         DBX222_6 : Bool;
         DBX222_7 : Bool;
         DBX223_0 : Bool;
         DBX223_1 : Bool;
         DBX223_2 : Bool;
         DBX223_3 : Bool;
         DBX223_4 : Bool;
         DBX223_5 : Bool;
         DBX223_6 : Bool;
         DBX223_7 : Bool;
         DBX224_0 : Bool;
         DBX224_1 : Bool;
         DBX224_2 : Bool;
         DBX224_3 : Bool;
         DBX224_4 : Bool;
         DBX224_5 : Bool;
         DBX224_6 : Bool;
         DBX224_7 : Bool;
         DBX225_0 : Bool;
         DBX225_1 : Bool;
         DBX225_2 : Bool;
         DBX225_3 : Bool;
         DBX225_4 : Bool;
         DBX225_5 : Bool;
         DBX225_6 : Bool;
         DBX225_7 : Bool;
         DBX226_0 : Bool;   // 9;CHAIN T7B;Stop Permisie Cuplare Lant T7-B Actionat;DI;A1;26;M;K
         DBX226_1 : Bool;   // 9;CHAIN T7B;TimeOut Cuplare/Decuplare Alim.Inv. Lant T7-B;DI;A1;26;M;O;K
         DBX226_2 : Bool;   // 9;CHAIN T7B;Lipsa Tensiune de Comanda Lant T7-B;DI;A1;26;M;K
         DBX226_3 : Bool;   // 9;CHAIN T7B;Sectionator Alim.Inv. Mot. Lant T7-B Decuplat;DI;A2;26;M;K
         DBX226_4 : Bool;   // 9;CHAIN T7B;Inverter Mot. Lant T7-B Avarie;DI;A2;26;M;O;K
         DBX226_5 : Bool;
         DBX226_6 : Bool;
         DBX226_7 : Bool;
         DBX227_0 : Bool;
         DBX227_1 : Bool;   // 9;CHAIN T7B;TimeOut Deplasare Lant T7-B in pozitia Pas;DI;A1;26;M;O;K
         DBX227_2 : Bool;   // 9;CHAIN T7B;Problema Contactor sau Prot. Termica Frana Lant T7-B;DI;A1;26;M;K
         DBX227_3 : Bool;   // 9;CHAIN T7B;TimeOut Deplasare Lant T7-B;DI;A1;26;M;O;K
         DBX227_4 : Bool;   // 9;CHAIN T7B;Disj. Termic Alim. Vent.Mot. Lant T7-B Declansat;DI;A1;26;M
         DBX227_5 : Bool;
         DBX227_6 : Bool;
         DBX227_7 : Bool;
         DBX228_0 : Bool;
         DBX228_1 : Bool;
         DBX228_2 : Bool;
         DBX228_3 : Bool;
         DBX228_4 : Bool;
         DBX228_5 : Bool;
         DBX228_6 : Bool;
         DBX228_7 : Bool;
         DBX229_0 : Bool;
         DBX229_1 : Bool;
         DBX229_2 : Bool;
         DBX229_3 : Bool;
         DBX229_4 : Bool;
         DBX229_5 : Bool;
         DBX229_6 : Bool;
         DBX229_7 : Bool;
         DBX230_0 : Bool;   // 9;FLIPPER2 T7B;Lipsa Tensiune Alimentare Aruncator 2 T7-B;DI;A1;26;M;K
         DBX230_1 : Bool;   // 9;FLIPPER2 T7B;TimeOut Deplasare Aruncator 2 T7-B in pozitia Sus;DI;A1;26;M;O
         DBX230_2 : Bool;   // 9;FLIPPER2 T7B;TimeOut Deplasare Aruncator 2 T7-B in pozitia Jos;DI;A1;26;M;O
         DBX230_3 : Bool;
         DBX230_4 : Bool;
         DBX230_5 : Bool;
         DBX230_6 : Bool;
         DBX230_7 : Bool;
         DBX231_0 : Bool;
         DBX231_1 : Bool;
         DBX231_2 : Bool;
         DBX231_3 : Bool;
         DBX231_4 : Bool;
         DBX231_5 : Bool;
         DBX231_6 : Bool;
         DBX231_7 : Bool;
         DBX232_0 : Bool;
         DBX232_1 : Bool;
         DBX232_2 : Bool;
         DBX232_3 : Bool;
         DBX232_4 : Bool;
         DBX232_5 : Bool;
         DBX232_6 : Bool;
         DBX232_7 : Bool;
         DBX233_0 : Bool;
         DBX233_1 : Bool;
         DBX233_2 : Bool;
         DBX233_3 : Bool;
         DBX233_4 : Bool;
         DBX233_5 : Bool;
         DBX233_6 : Bool;
         DBX233_7 : Bool;
         DBX234_0 : Bool;   // 9;COLLECTOR T7B;Disjunctor Termic Motor Colector T7-B;DI;A1;26;M
         DBX234_1 : Bool;   // 9;COLLECTOR T7B;TimeOut Deplasare Colector T7-B;DI;A1;26;M;O
         DBX234_2 : Bool;   // 9;COLLECTOR T7B;Disjunctor Termic Alim. Motor Colector T7-B;DI;A1;26;M
         DBX234_3 : Bool;   // 9;COLLECTOR T7B;Colector T7-B LB PLIN OFF;SQ;W3;26;O
         DBX234_4 : Bool;
         DBX234_5 : Bool;
         DBX234_6 : Bool;
         DBX234_7 : Bool;
         DBX235_0 : Bool;
         DBX235_1 : Bool;
         DBX235_2 : Bool;
         DBX235_3 : Bool;
         DBX235_4 : Bool;
         DBX235_5 : Bool;
         DBX235_6 : Bool;
         DBX235_7 : Bool;
         DBX236_0 : Bool;
         DBX236_1 : Bool;
         DBX236_2 : Bool;
         DBX236_3 : Bool;
         DBX236_4 : Bool;
         DBX236_5 : Bool;
         DBX236_6 : Bool;
         DBX236_7 : Bool;
         DBX237_0 : Bool;
         DBX237_1 : Bool;
         DBX237_2 : Bool;
         DBX237_3 : Bool;
         DBX237_4 : Bool;
         DBX237_5 : Bool;
         DBX237_6 : Bool;
         DBX237_7 : Bool;
         DBX238_0 : Bool;
         DBX238_1 : Bool;
         DBX238_2 : Bool;
         DBX238_3 : Bool;
         DBX238_4 : Bool;
         DBX238_5 : Bool;
         DBX238_6 : Bool;
         DBX238_7 : Bool;
         DBX239_0 : Bool;
         DBX239_1 : Bool;
         DBX239_2 : Bool;
         DBX239_3 : Bool;
         DBX239_4 : Bool;
         DBX239_5 : Bool;
         DBX239_6 : Bool;
         DBX239_7 : Bool;
         DBX240_0 : Bool;
         DBX240_1 : Bool;
         DBX240_2 : Bool;
         DBX240_3 : Bool;
         DBX240_4 : Bool;
         DBX240_5 : Bool;
         DBX240_6 : Bool;
         DBX240_7 : Bool;
         DBX241_0 : Bool;
         DBX241_1 : Bool;
         DBX241_2 : Bool;
         DBX241_3 : Bool;
         DBX241_4 : Bool;
         DBX241_5 : Bool;
         DBX241_6 : Bool;
         DBX241_7 : Bool;
         DBX242_0 : Bool;   // 9;ROLLS T7-C;Suma Disj. Termice Mot. C.Role T7-C Declansat;DI;A1;25;M;K
         DBX242_1 : Bool;   // 9;ROLLS T7-C;Sectionator Alim.Inv. Mot. C.Role T7-C Decuplat;DI;A2;25;M
         DBX242_2 : Bool;   // 9;ROLLS T7-C;Lipsa Tensiune de Comanda C.Role T7-C;DI;A1;25;M
         DBX242_3 : Bool;   // 9;ROLLS T7-C;TimeOut Rotire Role C.Role T7-C;DI;A1;25;M;O
         DBX242_4 : Bool;   // 9;ROLLS T7-C;Role T7-C TimeOut Teava ON;SQ;A1;25;O
         DBX242_5 : Bool;   // 9;ROLLS T7-C;Role T7-C TimeOut Teava SLOW;SQ;A1;25;O
         DBX242_6 : Bool;   // 9;ROLLS T7-C;Role T7-C TimeOut Pozitionare Teava;SQ;A1;25;O
         DBX242_7 : Bool;   // 9;ROLLS T7-C;Role T7-C TimeOut Teava OFF;SQ;A1;25;O
         DBX243_0 : Bool;
         DBX243_1 : Bool;
         DBX243_2 : Bool;
         DBX243_3 : Bool;
         DBX243_4 : Bool;   // 9;ROLLS T7-C;Disj. Termic Alim.Vent.Mot. C.Role T7-C - Declansat;DI;A1;25;M
         DBX243_5 : Bool;
         DBX243_6 : Bool;   // 9;ROLLS T7-C;Inverter Mot. C.Role T7-C - Avarie;DI;A1;25;M;O
         DBX243_7 : Bool;
         DBX244_0 : Bool;
         DBX244_1 : Bool;
         DBX244_2 : Bool;   // 9;ROLLS T7-C;Suma Disj. Th. Vent.Mot. C.Role T7-C - Declansat;DI;A1;25;M
         DBX244_3 : Bool;   // 9;ROLLS T7-C;TimeOut Cuplare/Decuplare Vent.Mot. C.Role T7-C;DI;A1;25;M;O
         DBX244_4 : Bool;   // 9;ROLLS T7-C;TimeOut Cuplare/Decuplare Alim.Inv. C.Role T7-C;DI;A1;25;M;O
         DBX244_5 : Bool;
         DBX244_6 : Bool;
         DBX244_7 : Bool;
         DBX245_0 : Bool;
         DBX245_1 : Bool;
         DBX245_2 : Bool;
         DBX245_3 : Bool;
         DBX245_4 : Bool;
         DBX245_5 : Bool;
         DBX245_6 : Bool;
         DBX245_7 : Bool;
         DBX246_0 : Bool;   // 9;FLIPPER T7-C;Lipsa Tensiune Alimentare Aruncator T7-C;DI;A1;25;M
         DBX246_1 : Bool;   // 9;FLIPPER T7-C;TimeOut Deplasare Aruncator T7-C in pozitia Sus;DI;A1;25;M;O
         DBX246_2 : Bool;   // 9;FLIPPER T7-C;TimeOut Deplasare Aruncator T7-C in pozitia Jos;DI;A1;25;M;O
         DBX246_3 : Bool;
         DBX246_4 : Bool;
         DBX246_5 : Bool;
         DBX246_6 : Bool;
         DBX246_7 : Bool;
         DBX247_0 : Bool;
         DBX247_1 : Bool;
         DBX247_2 : Bool;
         DBX247_3 : Bool;
         DBX247_4 : Bool;
         DBX247_5 : Bool;
         DBX247_6 : Bool;
         DBX247_7 : Bool;
         DBX248_0 : Bool;
         DBX248_1 : Bool;
         DBX248_2 : Bool;
         DBX248_3 : Bool;
         DBX248_4 : Bool;
         DBX248_5 : Bool;
         DBX248_6 : Bool;
         DBX248_7 : Bool;
         DBX249_0 : Bool;
         DBX249_1 : Bool;
         DBX249_2 : Bool;
         DBX249_3 : Bool;
         DBX249_4 : Bool;
         DBX249_5 : Bool;
         DBX249_6 : Bool;
         DBX249_7 : Bool;
         DBX250_0 : Bool;   // 9;COLLECTOR T7C;Disjunctor Termic Motor Colector T7-C;DI;A1;25;M
         DBX250_1 : Bool;   // 9;COLLECTOR T7C;TimeOut Deplasare Colector T7-C;DI;A1;25;M;O
         DBX250_2 : Bool;   // 9;COLLECTOR T7C;Disjunctor Termic Alim. Motor Colector T7-C;DI;A1;25;M
         DBX250_3 : Bool;   // 9;COLLECTOR T7C;Colector T7-C TimeOut Colector Plin;SQ;A1;25;O
         DBX250_4 : Bool;
         DBX250_5 : Bool;
         DBX250_6 : Bool;
         DBX250_7 : Bool;
         DBX251_0 : Bool;
         DBX251_1 : Bool;
         DBX251_2 : Bool;
         DBX251_3 : Bool;
         DBX251_4 : Bool;
         DBX251_5 : Bool;
         DBX251_6 : Bool;
         DBX251_7 : Bool;
         DBX252_0 : Bool;
         DBX252_1 : Bool;
         DBX252_2 : Bool;
         DBX252_3 : Bool;
         DBX252_4 : Bool;
         DBX252_5 : Bool;
         DBX252_6 : Bool;
         DBX252_7 : Bool;
         DBX253_0 : Bool;
         DBX253_1 : Bool;
         DBX253_2 : Bool;
         DBX253_3 : Bool;
         DBX253_4 : Bool;
         DBX253_5 : Bool;
         DBX253_6 : Bool;
         DBX253_7 : Bool;
         DBX254_0 : Bool;   // 9;TAMPON T7-C;Lipsa Tensiune Alimentare Tampon T7-C;DI;A1;25;M
         DBX254_1 : Bool;   // 9;TAMPON T7-C;TimeOut Deplasare Tampon T7-C in pozitia Sus;DI;A1;25;M;O
         DBX254_2 : Bool;   // 9;TAMPON T7-C;TimeOut Deplasare Tampon T7-C in pozitia Jos;DI;A1;25;M;O
         DBX254_3 : Bool;
         DBX254_4 : Bool;
         DBX254_5 : Bool;
         DBX254_6 : Bool;
         DBX254_7 : Bool;
         DBX255_0 : Bool;
         DBX255_1 : Bool;
         DBX255_2 : Bool;
         DBX255_3 : Bool;
         DBX255_4 : Bool;
         DBX255_5 : Bool;
         DBX255_6 : Bool;
         DBX255_7 : Bool;
         DBX256_0 : Bool;
         DBX256_1 : Bool;
         DBX256_2 : Bool;
         DBX256_3 : Bool;
         DBX256_4 : Bool;
         DBX256_5 : Bool;
         DBX256_6 : Bool;
         DBX256_7 : Bool;
         DBX257_0 : Bool;
         DBX257_1 : Bool;
         DBX257_2 : Bool;
         DBX257_3 : Bool;
         DBX257_4 : Bool;
         DBX257_5 : Bool;
         DBX257_6 : Bool;
         DBX257_7 : Bool;
         DBX258_0 : Bool;
         DBX258_1 : Bool;
         DBX258_2 : Bool;
         DBX258_3 : Bool;
         DBX258_4 : Bool;
         DBX258_5 : Bool;
         DBX258_6 : Bool;
         DBX258_7 : Bool;
         DBX259_0 : Bool;
         DBX259_1 : Bool;
         DBX259_2 : Bool;
         DBX259_3 : Bool;
         DBX259_4 : Bool;
         DBX259_5 : Bool;
         DBX259_6 : Bool;
         DBX259_7 : Bool;
         DBX260_0 : Bool;   // 9;DEBITARE;Disjunctor Termic Alim. Convertizor Lama;DI;A1;25;M
         DBX260_1 : Bool;   // 9;DEBITARE;TimeOut Cuplare/Decup. Cont. Convertizor Lama;DI;A1;25;M;O
         DBX260_2 : Bool;   // 9;DEBITARE;Disjunctor Termic Alim. Pompa Statie Hidraulica;DI;A2;25;M
         DBX260_3 : Bool;   // 9;DEBITARE;TimeOut Cuplare/Decup. Pompa Statie Hidraulica;DI;A1;25;M;O
         DBX260_4 : Bool;   // 9;DEBITARE;Disjunctor Termic Alim. Rezistenta Incalzire Ulei;DI;A1;25;M
         DBX260_5 : Bool;   // 9;DEBITARE;TimeOut Cuplare/Decup. Rezistenta Incalzire Ulei;DI;A1;25;M;O
         DBX260_6 : Bool;   // 9;DEBITARE;Disjunctor Termic Alim. Motor Vent. Statie Hidr.;DI;A1;25;M
         DBX260_7 : Bool;   // 9;DEBITARE;TimeOut Cuplare/Decup. Motor Vent. Statie Hidr.;DI;A1;25;M;O
         DBX261_0 : Bool;   // 9;DEBITARE;Disjunctor Termic Alim. Motor Pompa Racire Lama;DI;A1;25;M
         DBX261_1 : Bool;   // 9;DEBITARE;TimeOut Cuplare/Decup. Motor Pompa Racire Lama;DI;A1;25;M;O
         DBX261_2 : Bool;   // 9;DEBITARE;TimeOut Depl. Rola Singulara T7C in Pozitia 'Sus';DI;A1;25;M;O
         DBX261_3 : Bool;   // 9;DEBITARE;TimeOut Depl. Rola Singulara T7C in Pozitia 'Jos';DI;A1;25;M;O
         DBX261_4 : Bool;   // 9;DEBITARE;TimeOut Depl. Role T7C in Pozitia 'Sus';DI;A1;25;M;O
         DBX261_5 : Bool;   // 9;DEBITARE;TimeOut Depl. Role T7C in Pozitia 'Jos';DI;A1;25;M;O
         DBX261_6 : Bool;   // 9;DEBITARE;TimeOut Depl. Opritor Mobil in Pozitia 'Sus';DI;A1;25;M;O
         DBX261_7 : Bool;   // 9;DEBITARE;TimeOut Depl. Opritor Mobil in Pozitia 'Jos';DI;A1;25;M;O
         DBX262_0 : Bool;   // 9;DEBITARE;TimeOut Depl. Lama Circulara in Pozitia 'Sus';DI;A1;25;M;O
         DBX262_1 : Bool;   // 9;DEBITARE;TimeOut Depl. Lama Circulara in Pozitia 'Jos';DI;A1;25;M;O
         DBX262_2 : Bool;   // 9;DEBITARE;TimeOut Depl. Menghina in Pozitia 'Deschis';DI;A1;25;M;O
         DBX262_3 : Bool;   // 9;DEBITARE;Avertizare Coliziune Teava cu Rola Singulara T7C;DI;A1;25;O
         DBX262_4 : Bool;   // 9;DEBITARE;Avertizare Coliziune Teava cu Calea cu Role T7C;DI;A1;25;O
         DBX262_5 : Bool;   // 9;DEBITARE;Avertizare Coliziune Teava Opritor Mobil Masa T7C;DI;A1;25;O
         DBX262_6 : Bool;   // 9;DEBITARE;Avertizare Coliziune Teava cu Lama Circulara T7C;DI;A1;25;O
         DBX262_7 : Bool;   // 9;DEBITARE;Stare Convertizor - Avarie;DI;A1;25;M;O
         DBX263_0 : Bool;   // 9;DEBITARE;Disjuntor Termic Motor Lama Circulara - Declansat;DI;A1;25;M
         DBX263_1 : Bool;   // 9;DEBITARE;Nivel Apa Bazin Racire - Minim;DI;A1;25;M;O
         DBX263_2 : Bool;   // 9;DEBITARE;Temperatura Ulei Hidraulic - Minim;DI;W2;25;M;O
         DBX263_3 : Bool;   // 9;DEBITARE;Temperatura Ulei Hidraulic - Ridicat;DI;W2;25;M;O
         DBX263_4 : Bool;   // 9;DEBITARE;Temperatura Ulei Hidraulic - Maxim;DI;A1;25;M;O
         DBX263_5 : Bool;   // 9;DEBITARE;Nivel Ulei Hidraulic - Minim;DI;A1;25;M;O
         DBX263_6 : Bool;   // 9;DEBITARE;Releu Avarie (ciuperca) - Declansat;EM;A1;25;M;O;K
         DBX263_7 : Bool;
         DBX264_0 : Bool;   // 4;FIERASTRAU KASTO;Fierastrau Kasto Emergenta Apasata;EM;A1;11;M;O;K
         DBX264_1 : Bool;   // 4;FIERASTRAU KASTO;Avarie/Avertizare Fierastrau Kasto;DI;A1;11;M;O
         DBX264_2 : Bool;   // 4;FIERASTRAU KASTO;Pupitru Cabina Emergenta Apasata;EM;A1;11;M;O;K
         DBX264_3 : Bool;   // 4;TAMPON MASURARE PROBA;Disjunctor motor regl. proba decupl.;DI;A1;11;M
         DBX264_4 : Bool;   // 4;TAMPON MASURARE PROBA;Lipsa fbk cont linie mot. misc. inainte;DI;A1;11;M
         DBX264_5 : Bool;   // 4;TAMPON MASURARE PROBA;Lipsa fbk cont linie mot. misc. inapoi;DI;A1;11;M
         DBX264_6 : Bool;   // 4;ROLE KASTO;Disjunctor protectie ventilator motor 1 cuplat;DI;W2;11;M
         DBX264_7 : Bool;   // 4;ROLE KASTO;Confirmare cuplare contactor ventilator1 cuplat;DI;W2;11;M
         DBX265_0 : Bool;   // 4;ROLE KASTO;Disjunctor protectie ventilator motor 2 cuplat;DI;W2;11;M
         DBX265_1 : Bool;   // 4;ROLE KASTO;Confirmare cuplare contactor ventilator2 cuplat;DI;W2;11;M
         DBX265_2 : Bool;   // 4;ROLE KASTO;Disjunctor protectie ventilator motor 3 cuplat;DI;W2;11;M
         DBX265_3 : Bool;   // 4;ROLE KASTO;Confirmare cuplare contactor ventilator3 cuplat;DI;W2;11;M
         DBX265_4 : Bool;   // 4;ROLE KASTO;Disjunctor protectie ventilator motor 4 cuplat;DI;W2;11;M
         DBX265_5 : Bool;   // 4;ROLE KASTO;Confirmare cuplare contactor ventilator4 cuplat;DI;W2;11;M
         DBX265_6 : Bool;   // 4;ROLE KASTO;Disjunctor protectie ventilator motor 5 cuplat;DI;W2;11;M
         DBX265_7 : Bool;   // 4;ROLE KASTO;Confirmare cuplare contactor ventilator5 cuplat;DI;W2;11;M
         DBX266_0 : Bool;   // 4;ROLE KASTO;Disjunctor protectie ventilator motor 6 cuplat;DI;W2;11;M
         DBX266_1 : Bool;   // 4;ROLE KASTO;Confirmare cuplare contactor ventilator6 cuplat;DI;W2;11;M
         DBX266_2 : Bool;   // 4;ROLE KASTO;Disjunctor protectie ventilator motor 7 cuplat;DI;W2;11;M
         DBX266_3 : Bool;   // 4;ROLE KASTO;Confirmare cuplare contactor ventilator7 cuplat;DI;W2;11;M
         DBX266_4 : Bool;   // 4;ROLE KASTO;Disjunctor protectie ventilator motor 8 cuplat;DI;W2;11;M
         DBX266_5 : Bool;   // 4;ROLE KASTO;Confirmare cuplare contactor ventilator8 cuplat;DI;W2;11;M
         DBX266_6 : Bool;   // 4;ROLE KASTO;Disjunctor protectie ventilator motor 9 cuplat;DI;W2;11;M
         DBX266_7 : Bool;   // 4;ROLE KASTO;Confirmare cuplare contactor ventilator9 cuplat;DI;W2;11;M
         DBX267_0 : Bool;   // 4;ROLE KASTO;Disjunctor protectie ventilator motor 10 cuplat;DI;W2;11;M
         DBX267_1 : Bool;   // 4;ROLE KASTO;Confirmare cuplare contactor ventilat.10 cuplat;DI;W2;11;M
         DBX267_2 : Bool;   // 4;ROLE KASTO;Disjunctor protectie ventilator motor 11 cuplat;DI;W2;11;M
         DBX267_3 : Bool;   // 4;ROLE KASTO;Confirmare cuplare contactor ventilat.11 cuplat;DI;W2;11;M
         DBX267_4 : Bool;   // 4;ROLE KASTO;Disjunctor protectie ventilator motor 12 cuplat;DI;W2;11;M
         DBX267_5 : Bool;   // 4;ROLE KASTO;Confirmare cuplare contactor ventilat.12 cuplat;DI;W2;11;M
         DBX267_6 : Bool;   // 4;ROLE KASTO;Disjunctor protectie ventilator motor 13 cuplat;DI;W2;11;M
         DBX267_7 : Bool;   // 4;ROLE KASTO;Confirmare cuplare contactor ventilat.13 cuplat;DI;W2;11;M
         DBX268_0 : Bool;   // 4;ROLE KASTO;Disjunctor protectie ventilator motor 14 cuplat;DI;W2;11;M
         DBX268_1 : Bool;   // 4;ROLE KASTO;Confirmare cuplare contactor ventilat.14 cuplat;DI;W2;11;M
         DBX268_2 : Bool;   // 4;ROLE KASTO;Disjunctor protectie ventilator motor 15 cuplat;DI;W2;11;M
         DBX268_3 : Bool;   // 4;ROLE KASTO;Confirmare cuplare contactor ventilat.15 cuplat;DI;W2;11;M
         DBX268_4 : Bool;   // 4;ROLE KASTO;Fuzibil protectie convertizor;DI;A1;11;M
         DBX268_5 : Bool;   // 4;ROLE KASTO;Disjunctor monitorizare fuzibil convertizor;DI;A1;11;M
         DBX268_6 : Bool;   // 4;ROLE KASTO;Contactor alimentare convertizor;DI;A1;11;M
         DBX268_7 : Bool;   // 4;ROLE KASTO;Disjunctor protectie motoare;DI;A1;11;M
         DBX269_0 : Bool;   // 4;ROLE KASTO;Rola Mobila nu este ridicata;DI;A1;11;M
         DBX269_1 : Bool;
         DBX269_2 : Bool;
         DBX269_3 : Bool;
         DBX269_4 : Bool;
         DBX269_5 : Bool;
         DBX269_6 : Bool;
         DBX269_7 : Bool;
         DBX270_0 : Bool;   // 9;MARCARE;Disjunctor decuplat;DI;A2;24;M;K
         DBX270_1 : Bool;   // 9;MARCARE;Contactor ridicare decuplat;DI;A2;24;M;K
         DBX270_2 : Bool;   // 9;MARCARE;Contactor coborare decuplat;DI;A2;24;M;K
         DBX270_3 : Bool;   // 9;MARCARE;OCV camera fault;DI;A1;24;O
         DBX270_4 : Bool;   // 9;MARCARE;OCV alarma scor;DI;A1;24;O
         DBX270_5 : Bool;
         DBX270_6 : Bool;
         DBX270_7 : Bool;
         DBX271_0 : Bool;   // 4;FIERASTRAU KASTO;Citire atribute - Level 2 avarie generala;TK;W2;11;O
         DBX271_1 : Bool;   // 4;FIERASTRAU KASTO;Citire atribute - Destinatie plina;TK;W2;11;O
         DBX271_2 : Bool;   // 4;FIERASTRAU KASTO;Citire atribute - Sursa goala;TK;W2;11;O
         DBX271_3 : Bool;   // 4;FIERASTRAU KASTO;Incarca zona - Level 2 avarie generala;TK;W2;11;O
         DBX271_4 : Bool;   // 4;FIERASTRAU KASTO;Incarca zona - idTrackingItem invalid;TK;W2;11;O
         DBX271_5 : Bool;   // 4;FIERASTRAU KASTO;Incarca zona-Itemul nu e in prima pozitie;TK;W2;11;O
         DBX271_6 : Bool;   // 4;FIERASTRAU KASTO;Incarca zona - Destinatie plina;TK;W2;11;O
         DBX271_7 : Bool;   // 4;FIERASTRAU KASTO;Incarca zona - Sursa goala;TK;W2;11;O
         DBX272_0 : Bool;   // 4;FIERASTRAU KASTO;Verifica zona T4-2-Level2 avarie generala;TK;W2;11;O
         DBX272_1 : Bool;   // 4;FIERASTRAU KASTO;Descarca zona Kasto-Level2 avarie general;TK;W2;11;O
         DBX272_2 : Bool;   // 4;FIERASTRAU KASTO;Descarca zona Kasto - Destinatie plina;TK;W2;11;O
         DBX272_3 : Bool;   // 4;FIERASTRAU KASTO;Descarca zona Kasto - Sursa goala;TK;W2;11;O
         DBX272_4 : Bool;   // 4;FIERASTRAU KASTO;Verifica zona Kasto-Level2 avarie general;TK;W2;11;O
         DBX272_5 : Bool;   // 4;FIERASTRAU KASTO;Pat racire - Zona Kasto pachete diferite;TK;W2;11;O
         DBX272_6 : Bool;
         DBX272_7 : Bool;
         DBX273_0 : Bool;
         DBX273_1 : Bool;
         DBX273_2 : Bool;
         DBX273_3 : Bool;
         DBX273_4 : Bool;
         DBX273_5 : Bool;
         DBX273_6 : Bool;
         DBX273_7 : Bool;
         DBX274_0 : Bool;
         DBX274_1 : Bool;
         DBX274_2 : Bool;
         DBX274_3 : Bool;
         DBX274_4 : Bool;
         DBX274_5 : Bool;
         DBX274_6 : Bool;
         DBX274_7 : Bool;
         DBX275_0 : Bool;
         DBX275_1 : Bool;
         DBX275_2 : Bool;
         DBX275_3 : Bool;
         DBX275_4 : Bool;
         DBX275_5 : Bool;
         DBX275_6 : Bool;
         DBX275_7 : Bool;
         DBX276_0 : Bool;
         DBX276_1 : Bool;
         DBX276_2 : Bool;
         DBX276_3 : Bool;
         DBX276_4 : Bool;
         DBX276_5 : Bool;
         DBX276_6 : Bool;
         DBX276_7 : Bool;
         DBX277_0 : Bool;
         DBX277_1 : Bool;
         DBX277_2 : Bool;
         DBX277_3 : Bool;
         DBX277_4 : Bool;
         DBX277_5 : Bool;
         DBX277_6 : Bool;
         DBX277_7 : Bool;
         DBX278_0 : Bool;
         DBX278_1 : Bool;
         DBX278_2 : Bool;
         DBX278_3 : Bool;
         DBX278_4 : Bool;
         DBX278_5 : Bool;
         DBX278_6 : Bool;
         DBX278_7 : Bool;
         DBX279_0 : Bool;
         DBX279_1 : Bool;
         DBX279_2 : Bool;
         DBX279_3 : Bool;
         DBX279_4 : Bool;
         DBX279_5 : Bool;
         DBX279_6 : Bool;
         DBX279_7 : Bool;
         DBX280_0 : Bool;   // 1;Create Tracking;Time Out LEV2;TK;W2;1;O
         DBX280_1 : Bool;   // 1;New item load;Time Out LEV2;TK;W2;1;O
         DBX280_2 : Bool;   // 1;Item Count;Time Out LEV2;TK;W2;1;O
         DBX280_3 : Bool;   // 2;Check Product;Time Out LEV2;TK;W2;1;O
         DBX280_4 : Bool;   // 4;Check Product;Time Out LEV2;TK;W2;8;O
         DBX280_5 : Bool;   // 5;Create Tracking;Time Out LEV2;TK;W2;16;O
         DBX280_6 : Bool;   // 5;M5 Temper Entrance Check Product;Time Out LEV2;TK;W2;15;O
         DBX280_7 : Bool;   // 5;M5 Temper Entrance New Item Load;Time Out LEV2;TK;W2;15;O
         DBX281_0 : Bool;   // 5;M5 Temper Entrance Item Count;Time Out LEV2;TK;W2;15;O
         DBX281_1 : Bool;   // 6;M6 Temper Furnace Check Product;Time Out LEV2;TK;W2;15;O
         DBX281_2 : Bool;   // 8;M8 Straightening Check Product;Time Out LEV2;TK;W2;22;O
         DBX281_3 : Bool;   // 8;M8 Straightening New Item Load;Time Out LEV2;TK;W2;22;O
         DBX281_4 : Bool;   // 8;M8 Straightening New Item Count;Time Out LEV2;TK;W2;22;O
         DBX281_5 : Bool;   // 9;M9 Stamping Check Product;Time Out LEV2;TK;W2;23;O
         DBX281_6 : Bool;   // 9;M9 Stamping New Item Load;Time Out LEV2;TK;W2;23;O
         DBX281_7 : Bool;   // 9;M9 Stamping Item Count;Time Out LEV2;TK;W2;23;O
         DBX282_0 : Bool;   // 10;M10 Exit Check Product;Time Out LEV2;TK;W2;26;O
         DBX282_1 : Bool;   // 10;M10 Exit New Item Load;Time Out LEV2;TK;W2;26;O
         DBX282_2 : Bool;   // 10;M10 Exit New Item Count;Time Out LEV2;TK;W2;26;O
         DBX282_3 : Bool;   // 1;Z1 Entrance Quench Load;Time Out LEV2;TK;W2;1;O
         DBX282_4 : Bool;   // 3;Z3 Quenching Head Unload;Time Out LEV2;TK;W2;8;O
         DBX282_5 : Bool;   // 3;Z4 Exit Quench Unload;Time Out LEV2;TK;W2;10;O
         DBX282_6 : Bool;   // 4;Z5 Cool. Bench T4 load;Time Out LEV2;TK;W2;10;O
         DBX282_7 : Bool;   // 4;Z5 Cool. Bench T4 Exit Check;Time Out LEV2;TK;W2;10;O
         DBX283_0 : Bool;   // 4;Z5 Cool. Bench T4 Unload;Time Out LEV2;TK;W2;10;O
         DBX283_1 : Bool;   // 4;Z6 Exit T4 Get Pipe Attributes;Time Out LEV2;TK;W2;10;O
         DBX283_2 : Bool;   // 4;Z6 Exit T4 Unload;Time Out LEV2;TK;W2;14;O
         DBX283_3 : Bool;   // 4;Z8 Cool. Bench T5 Exit Load;Time Out LEV2;TK;W2;14;O
         DBX283_4 : Bool;   // 4;Z8 Cool. Bench T5 Exit Check;Time Out LEV2;TK;W2;14;O
         DBX283_5 : Bool;   // 4;Z8 Cool. Bench T5 Unload;Time Out LEV2;TK;W2;14;O
         DBX283_6 : Bool;   // 4;Z9 Exit T5 Get Pipe Attributes;Time Out LEV2;TK;W2;14;O
         DBX283_7 : Bool;   // 1;Z1 Entrance Quench Exit Check;Time Out LEV2;TK;W2;1;O
         DBX284_0 : Bool;   // 4;Z9 Exit T5 Unload;Time Out LEV2;TK;W2;15;O
         DBX284_1 : Bool;   // 4;Z10 Cool. Bench T6 Exit Load;Time Out LEV2;TK;W2;15;O
         DBX284_2 : Bool;   // 4;Z10 Cool. Bench T6 Exit Check;Time Out LEV2;TK;W2;15;O
         DBX284_3 : Bool;   // 4;Z10 Cool. Bench T6 Unload;Time Out LEV2;TK;W2;15;O
         DBX284_4 : Bool;   // 5;Z11 Entrance Temper Zone Load;Time Out LEV2;TK;W2;16;O
         DBX284_5 : Bool;   // 5;Z11 Entrance Temper Get Pipe Attributes;Time Out LEV2;TK;W2;15;O
         DBX284_6 : Bool;   // 7;Z13 Exit Temper Unload;Time Out LEV2;TK;W2;21;O
         DBX284_7 : Bool;   // 8;Z14 T7 Unload;Time Out LEV2;TK;W2;21;O
         DBX285_0 : Bool;   // 8;Z15 Straightening Unload;Time Out LEV2;TK;W2;22;O
         DBX285_1 : Bool;   // 8;Z16 T7A Loading Unload;Time Out LEV2;TK;W2;23;O
         DBX285_2 : Bool;   // 8;Z17 Cool.Bench T7A Exit Load;Time Out LEV2;TK;W2;23;O
         DBX285_3 : Bool;   // 8;Z17 Cool.Bench T7A Exit Check;Time Out LEV2;TK;W2;23;O
         DBX285_4 : Bool;   // 8;Z17 Cool.Bench T7A Unload;Time Out LEV2;TK;W2;23;O
         DBX285_5 : Bool;   // 9;Z18 Exit T7A Exit Check;Time Out LEV2;TK;W2;23;O
         DBX285_6 : Bool;   // 9;Z18 Exit T7A Unload;Time Out LEV2;TK;W2;26;O
         DBX285_7 : Bool;   // 9;Z18 Exit T7A Get Pipe Attributes;Time Out LEV2;TK;W2;23;O
         DBX286_0 : Bool;   // 9;Z19 Temper Sample Cut Load;Time Out LEV2;TK;W2;25;O
         DBX286_1 : Bool;   // 9;Z19 Temper Sample Cut Unload;Time Out LEV2;TK;W2;25;O
         DBX286_2 : Bool;   // 9;Z20 Cool.Bench T7B Exit Load;Time Out LEV2;TK;W2;26;O
         DBX286_3 : Bool;   // 9;Z20 Cool.Bench T7B Exit Check;Time Out LEV2;TK;W2;26;O
         DBX286_4 : Bool;   // 9;Z20 Cool.Bench T7B Unload;Time Out LEV2;TK;W2;26;O
         DBX286_5 : Bool;   // 9;Z21 Exit T7B Check;Time Out LEV2;TK;W2;26;O
         DBX286_6 : Bool;   // 9;Z21 Exit T7B Unload;Time Out LEV2;TK;W2;26;O
         DBX286_7 : Bool;   // 9;Send Data Stamping Machine;Time Out LEV2;TK;W2;23;O
         DBX287_0 : Bool;   // 8;Z14 T7 Exit Check;Time Out LEV2;TK;W2;21;O
         DBX287_1 : Bool;   // 3;Z3 Quenching Head Exit Check;Time Out LEV2;TK;W2;8;O
         DBX287_2 : Bool;   // 5;Z11 Temper Entrance Exit Check;Time Out LEV2;TK;W2;16;O
         DBX287_3 : Bool;   // 4;Z7 Quench Sample Unload;Time Out LEV2;TK;W2;12;O
         DBX287_4 : Bool;   // 4;Z23 Load T5 Zone Unload;Time Out LEV2;TK;W2;14;O
         DBX287_5 : Bool;   // 4;Z6 Exit T4 Load;Time Out LEV2;TK;W2;14;O
         DBX287_6 : Bool;   // 9;Z24 Load T7-B Zone Unload;Time Out LEV2;TK;W2;26;O
         DBX287_7 : Bool;   // 9;Z18 Exit T7-A Load;Time Out LEV2;TK;W2;23;O
         DBX288_0 : Bool;   // 9;Z24 Load T7-B Get Pipe Attributes;Time Out LEV2;TK;W2;26;O
         DBX288_1 : Bool;   // 4;Z6 Exit T4 Exit Check;Time Out LEV2;TK;W2;10;O
         DBX288_2 : Bool;   // 4;Z23 Load T5 Exit Check;Time Out LEV2;TK;W2;14;O
         DBX288_3 : Bool;   // 4;Z9 Exit T5 Exit Check;Time Out LEV2;TK;W2;14;O
         DBX288_4 : Bool;   // 9;Z24 Load T7B Exit Check;Time Out LEV2;TK;W2;26;O
         DBX288_5 : Bool;   // 8;Z17 Cool.Bench T7A Exit Check;Time Out LEV2;TK;W2;23;O
         DBX288_6 : Bool;   // 9;Z18 Sample Cut;Time Out LEV2;TK;W2;25;O
         DBX288_7 : Bool;   // 9;Z18 Sample Cut;Time Out LEV2;TK;W2;11;O
         DBX289_0 : Bool;
         DBX289_1 : Bool;
         DBX289_2 : Bool;
         DBX289_3 : Bool;
         DBX289_4 : Bool;
         DBX289_5 : Bool;
         DBX289_6 : Bool;
         DBX289_7 : Bool;
         DBX290_0 : Bool;   // 1;Z1 Entrance Quench;Date Tracking Incoerente;TK;W2;1;O
         DBX290_1 : Bool;   // 2;Z2 Quench Furnace;Date Tracking Incoerente;TK;W1;3;O
         DBX290_2 : Bool;   // 3;Z3 Quenching Head;Date Tracking Incoerente;TK;W1;8;O
         DBX290_3 : Bool;   // 4;Z4 Quench Exit;Date Tracking Incoerente;TK;W1;10;O
         DBX290_4 : Bool;   // 4;Z5 Cooling bench T4;Date Tracking Incoerente;TK;W1;10;O
         DBX290_5 : Bool;   // 4;Z6 Exit T4;Date Tracking Incoerente;TK;W1;10;O
         DBX290_6 : Bool;   // 4;Z7 Quench sample cut;Date Tracking Incoerente;TK;W1;11;O
         DBX290_7 : Bool;   // 4;Z8 Cooling bench T5;Date Tracking Incoerente;TK;W1;14;O
         DBX291_0 : Bool;   // 4;Z9 Exit T5;Date Tracking Incoerente;TK;W1;14;O
         DBX291_1 : Bool;   // 4;Z10 Cooling Bench T6;Date Tracking Incoerente;TK;W1;15;O
         DBX291_2 : Bool;   // 5;Z11 Temper Entrance;Date Tracking Incoerente;TK;W1;15;O
         DBX291_3 : Bool;   // 6;Z12 Temper Furnance;Date Tracking Incoerente;TK;W1;17;O
         DBX291_4 : Bool;   // 7;Z13 Exit Temper;Date Tracking Incoerente;TK;W2;21;O
         DBX291_5 : Bool;   // 7;Z14 T7;Date Tracking Incoerente;TK;W2;21;O
         DBX291_6 : Bool;   // 8;Z15 Straightening;Date Tracking Incoerente;TK;W1;22;O
         DBX291_7 : Bool;   // 9;Z16 Load T7-A;Date Tracking Incoerente;TK;W1;23;O
         DBX292_0 : Bool;   // 9;Z17 Cooling bench T7-A;Date Tracking Incoerente;TK;W1;23;O
         DBX292_1 : Bool;   // 9;Z18 Exit T7-A;Date Tracking Incoerente;TK;W1;23;O
         DBX292_2 : Bool;   // 10;Z19 Temper Sample Cut;Date Tracking Incoerente;TK;W1;25;O
         DBX292_3 : Bool;   // 10;Z20 Cooling bench T7-B;Date Tracking Incoerente;TK;W1;26;O
         DBX292_4 : Bool;   // 10;Z21 Exit T7-B;Date Tracking Incoerente;TK;W1;26;O
         DBX292_5 : Bool;   // 10;Z22 Exit;Date Tracking Incoerente;TK;W1;25;O
         DBX292_6 : Bool;   // 4;Z23 Load T5;Date Tracking Incoerente;TK;W1;14;O
         DBX292_7 : Bool;   // 9;Z24 Load T7-B;Date Tracking Incoerente;TK;W1;26;O
         DBX293_0 : Bool;
         DBX293_1 : Bool;
         DBX293_2 : Bool;
         DBX293_3 : Bool;
         DBX293_4 : Bool;
         DBX293_5 : Bool;
         DBX293_6 : Bool;
         DBX293_7 : Bool;
         DBX294_0 : Bool;   // 10;Z3 Exit T10 Get Pipe Attributes;Time Out LEV2;TK;W2;28;O
         DBX294_1 : Bool;   // 10;Z3 Exit T10 Exit Check;Time Out LEV2;TK;W2;28;O
         DBX294_2 : Bool;   // 10;Z26 Load RC01 T10 Unload;Time Out LEV2;TK;W2;28;O
         DBX294_3 : Bool;   // 10;Z26 Exit RC01 Exit Check;Time Out LEV2;TK;W2;28;O
         DBX294_4 : Bool;   // 10;Z27 Load Pat T10 Unload;Time Out LEV2;TK;W2;28;O
         DBX294_5 : Bool;   // 10;Z27 Exit Pat T10 Exit Check;Time Out LEV2;TK;W2;28;O
         DBX294_6 : Bool;   // 10;Z28 Load RC02 Pat T10 Unload;Time Out LEV2;TK;W2;28;O
         DBX294_7 : Bool;   // 10;Z28 Exit RC02 Exit Check;Time Out LEV2;TK;W2;28;O
         DBX295_0 : Bool;   // 10;Z25 Load Quence RC02 Unload;Time Out LEV2;TK;W2;28;O
         DBX295_1 : Bool;   // 10;Z19 T7-C Get Pipe Attributes;Time Out LEV2;TK;W2;28;O
         DBX295_2 : Bool;   // 9;Send Data Stamping Machine;Time Out LEV2;TK;W2;28;O
         DBX295_3 : Bool;   // 9;Send Data Stamping Machine Robot;Time Out LEV2;TK;W2;28;O
         DBX295_4 : Bool;
         DBX295_5 : Bool;
         DBX295_6 : Bool;
         DBX295_7 : Bool;
         DBX296_0 : Bool;
         DBX296_1 : Bool;
         DBX296_2 : Bool;
         DBX296_3 : Bool;
         DBX296_4 : Bool;
         DBX296_5 : Bool;
         DBX296_6 : Bool;
         DBX296_7 : Bool;
         DBX297_0 : Bool;
         DBX297_1 : Bool;
         DBX297_2 : Bool;
         DBX297_3 : Bool;
         DBX297_4 : Bool;
         DBX297_5 : Bool;
         DBX297_6 : Bool;
         DBX297_7 : Bool;
         DBX298_0 : Bool;   // 1;Create Tracking;Eroare Generala LEV2;TK;W2;1;O
         DBX298_1 : Bool;   // 1;Create Tracking;Cheie Inactiva in LEV2;TK;W2;1;O
         DBX298_2 : Bool;   // 1;Create Tracking;Lot Inactiv in LEV2;TK;W2;1;O
         DBX298_3 : Bool;   // 1;Create Tracking;Lipsa ID Tracking in LEV2;TK;W2;1;O
         DBX298_4 : Bool;   // 1;Create Tracking;ID deja existent in LEV2;TK;W2;1;O
         DBX298_5 : Bool;   // 1;New item load;Eroare Generala LEV2;TK;W2;1;O
         DBX298_6 : Bool;   // 1;New item load;Cheie Inactiva in LEV2;TK;W2;1;O
         DBX298_7 : Bool;   // 1;New item load;Lot Inactiv in LEV2;TK;W2;1;O
         DBX299_0 : Bool;   // 1;New item load;Lipsa ID Tracking in LEV2;TK;W2;1;O
         DBX299_1 : Bool;   // 1;New item load;ID Tracking deja existent in alt Lot;TK;W2;1;O
         DBX299_2 : Bool;   // 1;New item load;Eroare creare ID trecere;TK;W2;1;O
         DBX299_3 : Bool;   // 1;Item Count;Eroare Generala LEV2;TK;W2;1;O
         DBX299_4 : Bool;   // 1;Item Count;Lipsa ID Tracking in LEV2;TK;W2;1;O
         DBX299_5 : Bool;   // 2;Check Product;Eroare Generala LEV2;TK;W2;1;O
         DBX299_6 : Bool;   // 2;Check Product;Lipsa ID Tracking in LEV2;TK;W2;1;O
         DBX299_7 : Bool;   // 1;Z1 Entrance Quench Load;Eroare Generala LEV2;TK;W2;1;O
         DBX300_0 : Bool;   // 1;Z1 Entrance Quench Load;ID Invalid Tracking;TK;W2;1;O
         DBX300_1 : Bool;   // 1;Z1 Entrance Quench Load;Itemul Nu Este Primul;TK;W2;1;O
         DBX300_2 : Bool;   // 1;Z1 Entrance Quench Load;Zona Destinatie Plina;TK;W2;1;O
         DBX300_3 : Bool;   // 1;Z1 Entrance Quench Load;Eroare Incarcare Zona Goala;TK;W2;1;O
         DBX300_4 : Bool;   // 1;Z1 Entrance Quench Exit Check;Eroare Generala LEV2;TK;W2;1;O
         DBX300_5 : Bool;   // 1;Z1 Entrance Quench;Role T1-A Incoerenta Tracking;TK;W2;1;O
         DBX300_6 : Bool;   // 1;Z1 Entrance Quench;Role T1-C Incoerenta Tracking;TK;W2;2;O
         DBX300_7 : Bool;
         DBX301_0 : Bool;
         DBX301_1 : Bool;   // 1;Z1 Entrance Quench;Role T1-A SEQ.TRK Resetat;TK;W1;1;O
         DBX301_2 : Bool;   // 1;Z1 Entrance Quench;Role T1-C SEQ.TRK Resetat;TK;W1;2;O
         DBX301_3 : Bool;
         DBX301_4 : Bool;
         DBX301_5 : Bool;
         DBX301_6 : Bool;
         DBX301_7 : Bool;
         DBX302_0 : Bool;
         DBX302_1 : Bool;
         DBX302_2 : Bool;
         DBX302_3 : Bool;
         DBX302_4 : Bool;
         DBX302_5 : Bool;
         DBX302_6 : Bool;
         DBX302_7 : Bool;
         DBX303_0 : Bool;
         DBX303_1 : Bool;
         DBX303_2 : Bool;
         DBX303_3 : Bool;
         DBX303_4 : Bool;
         DBX303_5 : Bool;
         DBX303_6 : Bool;
         DBX303_7 : Bool;
         DBX304_0 : Bool;
         DBX304_1 : Bool;
         DBX304_2 : Bool;
         DBX304_3 : Bool;
         DBX304_4 : Bool;
         DBX304_5 : Bool;
         DBX304_6 : Bool;
         DBX304_7 : Bool;
         DBX305_0 : Bool;
         DBX305_1 : Bool;
         DBX305_2 : Bool;
         DBX305_3 : Bool;
         DBX305_4 : Bool;
         DBX305_5 : Bool;
         DBX305_6 : Bool;
         DBX305_7 : Bool;
         DBX306_0 : Bool;   // 3;Z3 Quenching Head Unload;Eroare Generala LEV2;TK;W2;8;O
         DBX306_1 : Bool;   // 3;Z3 Quenching Head Unload;Zona Destinatie Plina;TK;W2;8;O
         DBX306_2 : Bool;   // 3;Z3 Quenching Head Unload;Zona Sursa Goala;TK;W2;8;O
         DBX306_3 : Bool;   // 4;Check Product;Eroare Generala LEV2;TK;W2;8;O
         DBX306_4 : Bool;   // 4;Check Product;Lipsa ID Tracking in LEV2;TK;W2;8;O
         DBX306_5 : Bool;   // 3;Z3 Quenching Head Exit Check;Eroare Generala LEV2;TK;W2;8;O
         DBX306_6 : Bool;   // 3;Z3 Quenching Head;Role T4-1 Incoerenta Tracking;TK;W2;8;O
         DBX306_7 : Bool;
         DBX307_0 : Bool;   // 3;Z3 Quenching Head;Role T4-1 Seq Tracking Resetat;TK;W1;8;O
         DBX307_1 : Bool;
         DBX307_2 : Bool;
         DBX307_3 : Bool;
         DBX307_4 : Bool;
         DBX307_5 : Bool;
         DBX307_6 : Bool;
         DBX307_7 : Bool;
         DBX308_0 : Bool;
         DBX308_1 : Bool;
         DBX308_2 : Bool;
         DBX308_3 : Bool;
         DBX308_4 : Bool;
         DBX308_5 : Bool;
         DBX308_6 : Bool;
         DBX308_7 : Bool;
         DBX309_0 : Bool;
         DBX309_1 : Bool;
         DBX309_2 : Bool;
         DBX309_3 : Bool;
         DBX309_4 : Bool;
         DBX309_5 : Bool;
         DBX309_6 : Bool;
         DBX309_7 : Bool;
         DBX310_0 : Bool;   // 3;Z4 Exit Quench Unload;Eroare Generala LEV2;TK;W2;10;O
         DBX310_1 : Bool;   // 3;Z4 Exit Quench Unload;Zona Destinatie Plina;TK;W2;10;O
         DBX310_2 : Bool;   // 3;Z4 Exit Quench Unload;Zona Sursa Goala;TK;W2;10;O
         DBX310_3 : Bool;   // 4;Z5 Cool. Bench T4 Load;Excentric T4 Seq Tracking Resetat;TK;W1;10;O
         DBX310_4 : Bool;
         DBX310_5 : Bool;
         DBX310_6 : Bool;
         DBX310_7 : Bool;
         DBX311_0 : Bool;   // 3;Z3 Quenching Head Unload;Eroare Generala LEV2;TK;W2;28;O
         DBX311_1 : Bool;   // 3;Z3 Quenching Head Unload;Zona Destinatie Plina;TK;W2;28;O
         DBX311_2 : Bool;   // 3;Z3 Quenching Head Unload;Zona Sursa Goala;TK;W2;28;O
         DBX311_3 : Bool;   // 10;Check Product;Eroare Generala LEV2;TK;W2;28;O
         DBX311_4 : Bool;
         DBX311_5 : Bool;   // 10;Z26 Quenching Head Exit Check;Eroare Generala LEV2;TK;W2;28;O
         DBX311_6 : Bool;
         DBX311_7 : Bool;   // 10;Z26 Quenching Head;Role T10-1 Seq Tracking Resetat;TK;W1;28;O
         DBX312_0 : Bool;
         DBX312_1 : Bool;   // 10;Z26 Exit Quench Unload;Eroare Generala LEV2;TK;W2;28;O
         DBX312_2 : Bool;   // 10;Z26 Exit Quench Unload;Zona Destinatie Plina;TK;W2;28;O
         DBX312_3 : Bool;   // 10;Z27 Exit Quench Unload;Zona Sursa Goala;TK;W2;28;O
         DBX312_4 : Bool;   // 10;Z27 Cool. Bench T10 Load;Excentric T10 Seq Tracking Resetat;TK;W1;28;O
         DBX312_5 : Bool;
         DBX312_6 : Bool;   // 10;Z26 Cool. Bench T10 Exit Check;Eroare Generala LEV2;TK;W2;28;O
         DBX312_7 : Bool;   // 10;Z26 Cool. Bench T10;Role T10-2 Incoerenta Tracking;TK;W2;28;O
         DBX313_0 : Bool;   // 10;Z26 Cool. Bench T10 Unload;Eroare Generala LEV2;TK;W2;28;O
         DBX313_1 : Bool;   // 10;Z26 Cool. Bench T10 Unload;Zona Destinatie Plina;TK;W2;28;O
         DBX313_2 : Bool;   // 10;Z26 Cool. Bench T10 Unload;Zona Sursa Goala;TK;W2;28;O
         DBX313_3 : Bool;   // 10;Z26 Exit T10 Exit Check;Eroare Generala LEV2;TK;W2;28;O
         DBX313_4 : Bool;   // 10;Z26 Cool. Bench T10;STOPPER T10 Seq TRK Resetat;TK;W1;28;O
         DBX313_5 : Bool;   // 10;Z26 Exit T10 Exit Check;Zona Destinatie Plina;TK;W2;28O
         DBX313_6 : Bool;
         DBX313_7 : Bool;
         DBX314_0 : Bool;
         DBX314_1 : Bool;
         DBX314_2 : Bool;
         DBX314_3 : Bool;
         DBX314_4 : Bool;
         DBX314_5 : Bool;   // 4;Z5 Cool. Bench T4 Exit Check;Eroare Generala LEV2;TK;W2;10;O
         DBX314_6 : Bool;   // 4;Z5 Cool. Bench T4;Role T4-2 Incoerenta Tracking;TK;W2;10;O
         DBX314_7 : Bool;   // 4;Z5 Cool. Bench T4 Unload;Eroare Generala LEV2;TK;W2;10;O
         DBX315_0 : Bool;   // 4;Z5 Cool. Bench T4 Unload;Zona Destinatie Plina;TK;W2;10;O
         DBX315_1 : Bool;   // 4;Z5 Cool. Bench T4 Unload;Zona Sursa Goala;TK;W2;10;O
         DBX315_2 : Bool;   // 4;Z6 Exit T4 Exit Check;Eroare Generala LEV2;TK;W2;10;O
         DBX315_3 : Bool;
         DBX315_4 : Bool;   // 4;Z5 Cool. Bench T4;STOPPER T4 Seq TRK Resetat;TK;W1;10;O
         DBX315_5 : Bool;
         DBX315_6 : Bool;
         DBX315_7 : Bool;
         DBX316_0 : Bool;   // 10;Z27 Load Role T10-2;Incoerenta Tracking;TK;W2;O
         DBX316_1 : Bool;   // 10;Z27 Load Role T10-2 Exit;Rool T10-2 Seq TRK Resetat;TK;W1;O
         DBX316_2 : Bool;   // 10;Z27 Load Role T10-2 Zone Unload;Eroare Generala LEV2;TK;W2;O
         DBX316_3 : Bool;   // 10;Z27 Load Role T10-2 Zone Unload;Zona Destinatie Plina;TK;W2;O
         DBX316_4 : Bool;   // 10;Z24 Load Role T10-2 Zone Unload;Zona Sursa Goala;TK;W2;O
         DBX316_5 : Bool;   // 10;Z27 Load Role T10-2 Zone Check;Eroare Generala LEV2;TK;W2;O
         DBX316_6 : Bool;
         DBX316_7 : Bool;
         DBX317_0 : Bool;
         DBX317_1 : Bool;
         DBX317_2 : Bool;
         DBX317_3 : Bool;
         DBX317_4 : Bool;
         DBX317_5 : Bool;
         DBX317_6 : Bool;
         DBX317_7 : Bool;
         DBX318_0 : Bool;   // 4;Z6 Exit T4 Get Pipe Attributes;Eroare Generala LEV2;TK;W2;10;O
         DBX318_1 : Bool;   // 4;Z6 Exit T4 Get Pipe Attributes;Zona Destinatie Plina;TK;W2;10;O
         DBX318_2 : Bool;   // 4;Z6 Exit T4 Get Pipe Attributes;Zona Sursa Goala;TK;W2;10;O
         DBX318_3 : Bool;
         DBX318_4 : Bool;
         DBX318_5 : Bool;
         DBX318_6 : Bool;
         DBX318_7 : Bool;
         DBX319_0 : Bool;   // 9;Z24 Load T7-B Get Pipe Attributes;Eroare Generala LEV2;TK;W2;26;O
         DBX319_1 : Bool;   // 9;Z24 Load T7-B Get Pipe Attributes;Zona Destinatie Plina;TK;W2;26;O
         DBX319_2 : Bool;   // 9;Z24 Load T7-B Get Pipe Attributes;Zona Sursa Goala;TK;W2;26;O
         DBX319_3 : Bool;
         DBX319_4 : Bool;
         DBX319_5 : Bool;
         DBX319_6 : Bool;
         DBX319_7 : Bool;
         DBX320_0 : Bool;
         DBX320_1 : Bool;
         DBX320_2 : Bool;
         DBX320_3 : Bool;
         DBX320_4 : Bool;
         DBX320_5 : Bool;   // 4;Z23 Load T5 Exit;Rool T5-1 Seq TRK Resetat;TK;W1;14;O
         DBX320_6 : Bool;   // 9;Z24 Load T7-B;Incoerenta Tracking;TK;W2;26;O
         DBX320_7 : Bool;   // 4;Z23 Load T5 Exit Check;Eroare Generala LEV2;TK;W2;14;O
         DBX321_0 : Bool;   // 9;Z24 Load T7-B Zone Unload;Eroare Generala LEV2;TK;W2;26;O
         DBX321_1 : Bool;   // 9;Z24 Load T7-B Zone Unload;Zona Destinatie Plina;TK;W2;26;O
         DBX321_2 : Bool;   // 9;Z24 Load T7-B Zone Unload;Zona Sursa Goala;TK;W2;26;O
         DBX321_3 : Bool;   // 9;Z18 Exit T7-A Load;Eroare Generala LEV2;TK;W2;23;O
         DBX321_4 : Bool;   // 9;Z18 Exit T7-A Load;Item Tracking ID Invalid;TK;W2;23;O
         DBX321_5 : Bool;   // 9;Z18 Exit T7-A Load;Itemul Nu Este Primul;TK;W2;23;O
         DBX321_6 : Bool;   // 9;Z18 Exit T7-A Load;Zona Destinatie Plina;TK;W2;23;O
         DBX321_7 : Bool;   // 9;Z18 Exit T7-A Load;Incarcare Goala Nepermisa;TK;W2;23;O
         DBX322_0 : Bool;   // 4;Z23 Load T5 Zone Unload;Eroare Generala LEV2;TK;W2;14;O
         DBX322_1 : Bool;   // 4;Z23 Load T5 Zone Unload;Zona Destinatie Plina;TK;W2;14;O
         DBX322_2 : Bool;   // 4;Z23 Load T5 Zone Unload;Zona Sursa Goala;TK;W2;14;O
         DBX322_3 : Bool;   // 4;Z6 Exit T4 Load;Eroare Genrala LEV2;TK;W2;14;O
         DBX322_4 : Bool;   // 4;Z6 Exit T4 Load;Item Tracking ID Invalid;TK;W2;14;O
         DBX322_5 : Bool;   // 4;Z6 Exit T4 Load;Itemul Nu Este Primul;TK;W2;14;O
         DBX322_6 : Bool;   // 4;Z6 Exit T4 Load;Zona Destinatie Plina;TK;W2;14;O
         DBX322_7 : Bool;   // 4;Z6 Exit T4 Load;Incarcare Goala Nepermisa;TK;W2;14;O
         DBX323_0 : Bool;   // 4;Z23 Load T5;Incoerenta Tracking;TK;W2;14;O
         DBX323_1 : Bool;
         DBX323_2 : Bool;
         DBX323_3 : Bool;
         DBX323_4 : Bool;
         DBX323_5 : Bool;
         DBX323_6 : Bool;
         DBX323_7 : Bool;
         DBX324_0 : Bool;
         DBX324_1 : Bool;
         DBX324_2 : Bool;
         DBX324_3 : Bool;
         DBX324_4 : Bool;
         DBX324_5 : Bool;
         DBX324_6 : Bool;
         DBX324_7 : Bool;
         DBX325_0 : Bool;
         DBX325_1 : Bool;
         DBX325_2 : Bool;
         DBX325_3 : Bool;
         DBX325_4 : Bool;
         DBX325_5 : Bool;
         DBX325_6 : Bool;
         DBX325_7 : Bool;
         DBX326_0 : Bool;   // 4;Z7 Quench Sample Unload;Eroare Generala LEV2;TK;W2;12;O
         DBX326_1 : Bool;   // 4;Z7 Quench Sample Unload;Zona Destinatie Plina;TK;W2;12;O
         DBX326_2 : Bool;   // 4;Z7 Quench Sample Unload;Zona Sursa Goala;TK;W2;12;O
         DBX326_3 : Bool;
         DBX326_4 : Bool;
         DBX326_5 : Bool;
         DBX326_6 : Bool;
         DBX326_7 : Bool;
         DBX327_0 : Bool;
         DBX327_1 : Bool;
         DBX327_2 : Bool;
         DBX327_3 : Bool;
         DBX327_4 : Bool;
         DBX327_5 : Bool;
         DBX327_6 : Bool;
         DBX327_7 : Bool;
         DBX328_0 : Bool;
         DBX328_1 : Bool;
         DBX328_2 : Bool;
         DBX328_3 : Bool;
         DBX328_4 : Bool;
         DBX328_5 : Bool;
         DBX328_6 : Bool;
         DBX328_7 : Bool;
         DBX329_0 : Bool;
         DBX329_1 : Bool;
         DBX329_2 : Bool;
         DBX329_3 : Bool;
         DBX329_4 : Bool;
         DBX329_5 : Bool;
         DBX329_6 : Bool;
         DBX329_7 : Bool;   // 4;Z23 Load T5 Exit;Ex T5-1 Seq TRK Resetat;TK;W1;14;O
         DBX330_0 : Bool;   // 4;Z6 Exit T4 Unload;Eroare Generala LEV2;TK;W2;14;O
         DBX330_1 : Bool;   // 4;Z6 Exit T4 Unload;Zona Destinatie Plina;TK;W2;14;O
         DBX330_2 : Bool;   // 4;Z6 Exit T4 Unload;Zona Sursa Goala;TK;W2;14;O
         DBX330_3 : Bool;
         DBX330_4 : Bool;
         DBX330_5 : Bool;
         DBX330_6 : Bool;
         DBX330_7 : Bool;
         DBX331_0 : Bool;
         DBX331_1 : Bool;
         DBX331_2 : Bool;
         DBX331_3 : Bool;
         DBX331_4 : Bool;
         DBX331_5 : Bool;
         DBX331_6 : Bool;
         DBX331_7 : Bool;
         DBX332_0 : Bool;
         DBX332_1 : Bool;
         DBX332_2 : Bool;
         DBX332_3 : Bool;
         DBX332_4 : Bool;
         DBX332_5 : Bool;
         DBX332_6 : Bool;
         DBX332_7 : Bool;
         DBX333_0 : Bool;
         DBX333_1 : Bool;
         DBX333_2 : Bool;
         DBX333_3 : Bool;
         DBX333_4 : Bool;
         DBX333_5 : Bool;
         DBX333_6 : Bool;
         DBX333_7 : Bool;
         DBX334_0 : Bool;
         DBX334_1 : Bool;
         DBX334_2 : Bool;
         DBX334_3 : Bool;
         DBX334_4 : Bool;
         DBX334_5 : Bool;
         DBX334_6 : Bool;   // 4;Z8 Cool. Bench T5 Exit Check;Eroare Generala LEV2;TK;W2;14;O
         DBX334_7 : Bool;   // 4;Z8 Cool. Bench T5;Role T5-2 Incoerenta Tracking;TK;W2;14;O
         DBX335_0 : Bool;   // 4;Z8 Cool. Bench T5 Unload;Eroare Generala LEV2;TK;W2;14;O
         DBX335_1 : Bool;   // 4;Z8 Cool. Bench T5 Unload;Zona Destinatie Plina;TK;W2;14;O
         DBX335_2 : Bool;   // 4;Z8 Cool. Bench T5 Unload;Zona Sursa Goala;TK;W2;14;O
         DBX335_3 : Bool;   // 4;Z9 Exit T5 Exit Check;Eroare Generala LEV2;TK;W2;14;O
         DBX335_4 : Bool;   // 4;Z8 Cool. Bench T5;Opritor T5 Seq TRK Resetata;TK;W1;14;O
         DBX335_5 : Bool;
         DBX335_6 : Bool;
         DBX335_7 : Bool;
         DBX336_0 : Bool;
         DBX336_1 : Bool;
         DBX336_2 : Bool;
         DBX336_3 : Bool;
         DBX336_4 : Bool;
         DBX336_5 : Bool;
         DBX336_6 : Bool;
         DBX336_7 : Bool;
         DBX337_0 : Bool;
         DBX337_1 : Bool;
         DBX337_2 : Bool;
         DBX337_3 : Bool;
         DBX337_4 : Bool;
         DBX337_5 : Bool;
         DBX337_6 : Bool;
         DBX337_7 : Bool;
         DBX338_0 : Bool;
         DBX338_1 : Bool;   // 4;Z9 Exit T5 Get Pipe Attributes;Eroare Generala LEV2;TK;W2;14;O
         DBX338_2 : Bool;   // 4;Z9 Exit T5 Get Pipe Attributes;Zona Destinatie Plina;TK;W2;14;O
         DBX338_3 : Bool;   // 4;Z9 Exit T5 Get Pipe Attributes;Zona Sursa Goala;TK;W2;14;O
         DBX338_4 : Bool;
         DBX338_5 : Bool;
         DBX338_6 : Bool;
         DBX338_7 : Bool;
         DBX339_0 : Bool;
         DBX339_1 : Bool;
         DBX339_2 : Bool;
         DBX339_3 : Bool;
         DBX339_4 : Bool;
         DBX339_5 : Bool;
         DBX339_6 : Bool;
         DBX339_7 : Bool;
         DBX340_0 : Bool;
         DBX340_1 : Bool;
         DBX340_2 : Bool;
         DBX340_3 : Bool;
         DBX340_4 : Bool;
         DBX340_5 : Bool;
         DBX340_6 : Bool;
         DBX340_7 : Bool;
         DBX341_0 : Bool;
         DBX341_1 : Bool;
         DBX341_2 : Bool;
         DBX341_3 : Bool;
         DBX341_4 : Bool;
         DBX341_5 : Bool;
         DBX341_6 : Bool;
         DBX341_7 : Bool;
         DBX342_0 : Bool;
         DBX342_1 : Bool;
         DBX342_2 : Bool;
         DBX342_3 : Bool;
         DBX342_4 : Bool;
         DBX342_5 : Bool;
         DBX342_6 : Bool;
         DBX342_7 : Bool;
         DBX343_0 : Bool;
         DBX343_1 : Bool;
         DBX343_2 : Bool;
         DBX343_3 : Bool;
         DBX343_4 : Bool;
         DBX343_5 : Bool;
         DBX343_6 : Bool;
         DBX343_7 : Bool;
         DBX344_0 : Bool;
         DBX344_1 : Bool;
         DBX344_2 : Bool;
         DBX344_3 : Bool;
         DBX344_4 : Bool;
         DBX344_5 : Bool;
         DBX344_6 : Bool;
         DBX344_7 : Bool;
         DBX345_0 : Bool;
         DBX345_1 : Bool;
         DBX345_2 : Bool;
         DBX345_3 : Bool;
         DBX345_4 : Bool;
         DBX345_5 : Bool;
         DBX345_6 : Bool;
         DBX345_7 : Bool;
         DBX346_0 : Bool;   // 4;Z9 Exit T5;Excentric T6 Seq TRK Resetata;TK;W1;14;O
         DBX346_1 : Bool;   // 4;Z9 Exit T5 Unload;Eroare Generala LEV2;TK;W2;14;O
         DBX346_2 : Bool;   // 4;Z9 Exit T5 Unload;Zona Destinatie Plina;TK;W2;14;O
         DBX346_3 : Bool;   // 4;Z9 Exit T5 Unload;Zona Sursa Goala;TK;W2;14;O
         DBX346_4 : Bool;
         DBX346_5 : Bool;
         DBX346_6 : Bool;
         DBX346_7 : Bool;
         DBX347_0 : Bool;
         DBX347_1 : Bool;
         DBX347_2 : Bool;
         DBX347_3 : Bool;
         DBX347_4 : Bool;
         DBX347_5 : Bool;
         DBX347_6 : Bool;
         DBX347_7 : Bool;
         DBX348_0 : Bool;
         DBX348_1 : Bool;
         DBX348_2 : Bool;
         DBX348_3 : Bool;
         DBX348_4 : Bool;
         DBX348_5 : Bool;
         DBX348_6 : Bool;
         DBX348_7 : Bool;
         DBX349_0 : Bool;
         DBX349_1 : Bool;
         DBX349_2 : Bool;
         DBX349_3 : Bool;
         DBX349_4 : Bool;
         DBX349_5 : Bool;
         DBX349_6 : Bool;
         DBX349_7 : Bool;
         DBX350_0 : Bool;   // 4;Z10 Cool. Bench T6;Opritor T6 Seq TRK Resetata;TK;W1;15;O
         DBX350_1 : Bool;
         DBX350_2 : Bool;
         DBX350_3 : Bool;
         DBX350_4 : Bool;
         DBX350_5 : Bool;
         DBX350_6 : Bool;   // 4;Z10 Cool. Bench T6 Exit Check;Eroare Generala LEV2;TK;W2;15;O
         DBX350_7 : Bool;   // 4;Z10 Cool. Bench T6;Role T6 Incoerenta Tracking;TK;W2;15;O
         DBX351_0 : Bool;   // 4;Z10 Cool. Bench T6 Unload;Eroare Generala LEV2;TK;W2;15;O
         DBX351_1 : Bool;   // 4;Z10 Cool. Bench T6 Unload;Zona Destinatie Plina;TK;W2;15;O
         DBX351_2 : Bool;   // 4;Z10 Cool. Bench T6 Unload;Zona Sursa Goala;TK;W2;15;O
         DBX351_3 : Bool;   // 4;Z10 Cool. Bench T6;T1-D Incoerenta Tracking;TK;W2;15;O
         DBX351_4 : Bool;   // 5;Z11 Temper Entrance Exit Check;Eroare Generala LEV2;TK;W2;16;O
         DBX351_5 : Bool;
         DBX351_6 : Bool;
         DBX351_7 : Bool;
         DBX352_0 : Bool;
         DBX352_1 : Bool;
         DBX352_2 : Bool;
         DBX352_3 : Bool;
         DBX352_4 : Bool;
         DBX352_5 : Bool;
         DBX352_6 : Bool;
         DBX352_7 : Bool;
         DBX353_0 : Bool;
         DBX353_1 : Bool;
         DBX353_2 : Bool;
         DBX353_3 : Bool;
         DBX353_4 : Bool;
         DBX353_5 : Bool;
         DBX353_6 : Bool;
         DBX353_7 : Bool;
         DBX354_0 : Bool;
         DBX354_1 : Bool;   // 5;Z11 Entrance Temper Get Pipe Attributes;Eroare Gen.LEV2;TK;W2;15;O
         DBX354_2 : Bool;   // 5;Z11 Entrance Temper Get Pipe Attributes;Zona Destinatie Plin;TK;W2;15;O
         DBX354_3 : Bool;   // 5;Z11 Entrance Temper Get Pipe Attributes;Zona Sursa Goala;TK;W2;15;O
         DBX354_4 : Bool;   // 5;M5 Temper Entrance Check Product;Eroare Generala LEV2;TK;W2;15;O
         DBX354_5 : Bool;   // 5;M5 Temper Entrance Check Product;Lipsa ID Tracking LEV2;TK;W2;15;O
         DBX354_6 : Bool;
         DBX354_7 : Bool;
         DBX355_0 : Bool;
         DBX355_1 : Bool;
         DBX355_2 : Bool;
         DBX355_3 : Bool;
         DBX355_4 : Bool;
         DBX355_5 : Bool;
         DBX355_6 : Bool;
         DBX355_7 : Bool;
         DBX356_0 : Bool;
         DBX356_1 : Bool;
         DBX356_2 : Bool;
         DBX356_3 : Bool;
         DBX356_4 : Bool;
         DBX356_5 : Bool;
         DBX356_6 : Bool;
         DBX356_7 : Bool;
         DBX357_0 : Bool;
         DBX357_1 : Bool;
         DBX357_2 : Bool;
         DBX357_3 : Bool;
         DBX357_4 : Bool;
         DBX357_5 : Bool;
         DBX357_6 : Bool;
         DBX357_7 : Bool;
         DBX358_0 : Bool;
         DBX358_1 : Bool;
         DBX358_2 : Bool;
         DBX358_3 : Bool;
         DBX358_4 : Bool;
         DBX358_5 : Bool;
         DBX358_6 : Bool;
         DBX358_7 : Bool;
         DBX359_0 : Bool;
         DBX359_1 : Bool;
         DBX359_2 : Bool;
         DBX359_3 : Bool;
         DBX359_4 : Bool;
         DBX359_5 : Bool;
         DBX359_6 : Bool;
         DBX359_7 : Bool;
         DBX360_0 : Bool;
         DBX360_1 : Bool;
         DBX360_2 : Bool;
         DBX360_3 : Bool;
         DBX360_4 : Bool;
         DBX360_5 : Bool;
         DBX360_6 : Bool;
         DBX360_7 : Bool;
         DBX361_0 : Bool;
         DBX361_1 : Bool;
         DBX361_2 : Bool;
         DBX361_3 : Bool;
         DBX361_4 : Bool;
         DBX361_5 : Bool;
         DBX361_6 : Bool;
         DBX361_7 : Bool;
         DBX362_0 : Bool;
         DBX362_1 : Bool;   // 5;Create Tracking;Eroare Generala LEV2;TK;W2;16;O
         DBX362_2 : Bool;   // 5;Create Tracking;Cheie Inactiva in LEV2;TK;W2;16;O
         DBX362_3 : Bool;   // 5;Create Tracking;Lot Inactivin LEV2;TK;W2;16;O
         DBX362_4 : Bool;   // 5;Create Tracking;Lipsa ID Tracking in LEV2;TK;W2;16;O
         DBX362_5 : Bool;   // 5;Create Tracking;ID Deja Existent in LEV2;TK;W2;16;O
         DBX362_6 : Bool;   // 5;M5 Temper Entrance New Item Load;Eroare Generala LEV2;TK;W2;15;O
         DBX362_7 : Bool;   // 5;M5 Temper Entrance New Item Load;Cheie Inactiva in LEV2;TK;W2;15;O
         DBX363_0 : Bool;   // 5;M5 Temper Entrance New Item Load;Lot Inactiv in LEV2;TK;W2;15;O
         DBX363_1 : Bool;   // 5;M5 Temper Entrance New Item Load;Lipsa ID Tracking in LEV2;TK;W2;15;O
         DBX363_2 : Bool;   // 5;M5 Temper Entrance New Item Load;ID Track. Apartin Altui lot;TK;W2;15;O
         DBX363_3 : Bool;   // 5;M5 Temper Entrance New Item Load;Eroare Creare Pass Tracking;TK;W2;15;O
         DBX363_4 : Bool;   // 5;M5 Temper Entrance Item Count;Eroare Generala LEV2;TK;W2;15;O
         DBX363_5 : Bool;   // 5;M5 Temper Entrance Item Count;Lipsa ID Tracking LEV2;TK;W2;15;O
         DBX363_6 : Bool;   // 6;M6 Temper Furnace Check Product;Eroare Generala LEV2;TK;W2;15;O
         DBX363_7 : Bool;   // 6;M6 Temper Furnace Check Product;Lipsa ID Tracking LEV2;TK;W2;15;O
         DBX364_0 : Bool;   // 5;Z11 Entrance Temper Zone Load;Eroare Generala LEV2;TK;W2;16;O
         DBX364_1 : Bool;   // 5;Z11 Entrance Temper Zone Load;Item Tracking ID Invalid;TK;W2;16;O
         DBX364_2 : Bool;   // 5;Z11 Entrance Temper Zone Load;Itemul Nu Este Primul;TK;W2;16;O
         DBX364_3 : Bool;   // 5;Z11 Entrance Temper Zone Load;Zona Destinatie Plina;TK;W2;16;O
         DBX364_4 : Bool;   // 5;Z11 Entrance Temper Zone Load;Incarcare Goala Nepermisa;TK;W2;16;O
         DBX364_5 : Bool;   // 5;Z11 Entrance Temper Exit Check;Eroare Generala LEV2;TK;W2;16;O
         DBX364_6 : Bool;
         DBX364_7 : Bool;
         DBX365_0 : Bool;
         DBX365_1 : Bool;
         DBX365_2 : Bool;
         DBX365_3 : Bool;
         DBX365_4 : Bool;
         DBX365_5 : Bool;
         DBX365_6 : Bool;
         DBX365_7 : Bool;
         DBX366_0 : Bool;
         DBX366_1 : Bool;
         DBX366_2 : Bool;
         DBX366_3 : Bool;
         DBX366_4 : Bool;
         DBX366_5 : Bool;
         DBX366_6 : Bool;
         DBX366_7 : Bool;
         DBX367_0 : Bool;
         DBX367_1 : Bool;
         DBX367_2 : Bool;
         DBX367_3 : Bool;
         DBX367_4 : Bool;
         DBX367_5 : Bool;
         DBX367_6 : Bool;
         DBX367_7 : Bool;
         DBX368_0 : Bool;
         DBX368_1 : Bool;
         DBX368_2 : Bool;
         DBX368_3 : Bool;
         DBX368_4 : Bool;
         DBX368_5 : Bool;
         DBX368_6 : Bool;
         DBX368_7 : Bool;
         DBX369_0 : Bool;
         DBX369_1 : Bool;
         DBX369_2 : Bool;
         DBX369_3 : Bool;
         DBX369_4 : Bool;
         DBX369_5 : Bool;
         DBX369_6 : Bool;
         DBX369_7 : Bool;
         DBX370_0 : Bool;
         DBX370_1 : Bool;   // 7;Z13 Exit Temper Unload;Eroare Generala LEV2;TK;W2;21;O
         DBX370_2 : Bool;   // 7;Z13 Exit Temper Unload;Zona Destinatie Plina;TK;W2;21;O
         DBX370_3 : Bool;   // 7;Z13 Exit Temper Unload;Zona Sursa Goala;TK;W2;21;O
         DBX370_4 : Bool;
         DBX370_5 : Bool;
         DBX370_6 : Bool;
         DBX370_7 : Bool;
         DBX371_0 : Bool;
         DBX371_1 : Bool;   // 9;Z18 Exit T7A Exit Check;Eroare Generala LEV2;TK;W2;23;O
         DBX371_2 : Bool;   // 9;Z24 Load T7B Exit Check;Eroare Generala LEV2;TK;W2;26;O
         DBX371_3 : Bool;   // 9;Z19 Temper Sample Cut Load;Eroare Generala LEV2;TK;W2;25;O
         DBX371_4 : Bool;   // 9;Z19 Temper Sample Cut Load;Item Tracking ID Invalid;TK;W2;25;O
         DBX371_5 : Bool;   // 9;Z19 Temper Sample Cut Load;Itemul Nu Este Primul;TK;W2;25;O
         DBX371_6 : Bool;   // 9;Z19 Temper Sample Cut Load;Zona Destinatie Plina;TK;W2;25;O
         DBX371_7 : Bool;   // 9;Z19 Temper Sample Cut Load;Incarcare Goala Nepermisa;TK;W2;25;O
         DBX372_0 : Bool;   // 9;Z19 Temper Sample Cut Unload;Eroare Generala LEV2;TK;W2;25;O
         DBX372_1 : Bool;   // 9;Z19 Temper Sample Cut Unload;Zona Destinatie Plina;TK;W2;25;O
         DBX372_2 : Bool;   // 9;Z19 Temper Sample Cut Unload;Zona Sursa Goala;TK;W2;25;O
         DBX372_3 : Bool;   // 9;Z18 Exit T7A Unload;Eroare Generala LEV2;TK;W2;23;O
         DBX372_4 : Bool;   // 9;Z18 Exit T7A Unload;Zona Destinatie Plina;TK;W2;23;O
         DBX372_5 : Bool;   // 9;Z18 Exit T7A Unload;Zona Sursa Goala;TK;W2;23;O
         DBX372_6 : Bool;
         DBX372_7 : Bool;
         DBX373_0 : Bool;
         DBX373_1 : Bool;
         DBX373_2 : Bool;
         DBX373_3 : Bool;   // 9;Z20 Cool.Bench T7B Exit Check;Eroare Generala LEV2;TK;W2;26;O
         DBX373_4 : Bool;
         DBX373_5 : Bool;   // 9;Z20 Cool.Bench T7B Unload;Eroare Generala LEV2;TK;W2;26;O
         DBX373_6 : Bool;   // 9;Z20 Cool.Bench T7B Unload;Zona Destinatie Plina;TK;W2;26;O
         DBX373_7 : Bool;   // 9;Z20 Cool.Bench T7B Unload;Zona Sursa Goala;TK;W2;26;O
         DBX374_0 : Bool;   // 10;M10 Exit Check Product;Eroare Generala LEV2;TK;W2;26;O
         DBX374_1 : Bool;   // 10;M10 Exit Check Product;Lipsa ID Tracking in LEV2;TK;W2;26;O
         DBX374_2 : Bool;   // 10;M10 Exit New Item Load;Eroare Generala LEV2;TK;W2;26;O
         DBX374_3 : Bool;   // 10;M10 Exit New Item Load;Cheie Inactiva in LEV2;TK;W2;26;O
         DBX374_4 : Bool;   // 10;M10 Exit New Item Load;Lot Inactiv in LEV2;TK;W2;26;O
         DBX374_5 : Bool;   // 10;M10 Exit New Item Load;Lipsa ID Tracking in LEV2;TK;W2;26;O
         DBX374_6 : Bool;   // 10;M10 Exit New Item Load;ID Tracking Apartine Altui Lot;TK;W2;26;O
         DBX374_7 : Bool;   // 10;M10 Exit New Item Load;Eroare la Creare Tracking Pass;TK;W2;26;O
         DBX375_0 : Bool;   // 10;M10 Exit New Item Count;Eroare Generala LEV2;TK;W2;26;O
         DBX375_1 : Bool;   // 10;M10 Exit New Item Count;Lipsa ID Tracking in LEV2;TK;W2;26;O
         DBX375_2 : Bool;
         DBX375_3 : Bool;
         DBX375_4 : Bool;
         DBX375_5 : Bool;
         DBX375_6 : Bool;
         DBX375_7 : Bool;
         DBX376_0 : Bool;
         DBX376_1 : Bool;
         DBX376_2 : Bool;
         DBX376_3 : Bool;
         DBX376_4 : Bool;
         DBX376_5 : Bool;
         DBX376_6 : Bool;
         DBX376_7 : Bool;
         DBX377_0 : Bool;
         DBX377_1 : Bool;
         DBX377_2 : Bool;
         DBX377_3 : Bool;
         DBX377_4 : Bool;
         DBX377_5 : Bool;
         DBX377_6 : Bool;
         DBX377_7 : Bool;
         DBX378_0 : Bool;
         DBX378_1 : Bool;
         DBX378_2 : Bool;
         DBX378_3 : Bool;
         DBX378_4 : Bool;
         DBX378_5 : Bool;
         DBX378_6 : Bool;
         DBX378_7 : Bool;
         DBX379_0 : Bool;
         DBX379_1 : Bool;
         DBX379_2 : Bool;
         DBX379_3 : Bool;
         DBX379_4 : Bool;
         DBX379_5 : Bool;
         DBX379_6 : Bool;   // 8;Z14 T7 Exit Check;Eroare Generala LEV2;TK;W2;21;O
         DBX379_7 : Bool;   // 8;Z14 T7 Exit;SUTTON Incoerenta Tracking;TK;W2;21;O
         DBX380_0 : Bool;
         DBX380_1 : Bool;
         DBX380_2 : Bool;
         DBX380_3 : Bool;
         DBX380_4 : Bool;
         DBX380_5 : Bool;
         DBX380_6 : Bool;
         DBX380_7 : Bool;
         DBX381_0 : Bool;
         DBX381_1 : Bool;
         DBX381_2 : Bool;
         DBX381_3 : Bool;
         DBX381_4 : Bool;
         DBX381_5 : Bool;
         DBX381_6 : Bool;
         DBX381_7 : Bool;
         DBX382_0 : Bool;
         DBX382_1 : Bool;   // 8;Z15 Straightening Unload;Eroare Generala LEV2;TK;W2;22;O
         DBX382_2 : Bool;   // 8;Z15 Straightening Unload;Zona Destinatie Plina;TK;W2;22;O
         DBX382_3 : Bool;   // 8;Z15 Straightening Unload;Zona Sursa Goala;TK;W2;22;O
         DBX382_4 : Bool;   // 8;Z17 Cool.Bench T7A ;Load T7A Incoerenta Tracking;TK;W2;23;O
         DBX382_5 : Bool;   // 8;Z17 Cool.Bench T7A Exit Check;Eroare Generala LEV2;TK;W2;23;O
         DBX382_6 : Bool;
         DBX382_7 : Bool;
         DBX383_0 : Bool;
         DBX383_1 : Bool;
         DBX383_2 : Bool;
         DBX383_3 : Bool;
         DBX383_4 : Bool;
         DBX383_5 : Bool;
         DBX383_6 : Bool;
         DBX383_7 : Bool;
         DBX384_0 : Bool;
         DBX384_1 : Bool;
         DBX384_2 : Bool;
         DBX384_3 : Bool;
         DBX384_4 : Bool;
         DBX384_5 : Bool;
         DBX384_6 : Bool;
         DBX384_7 : Bool;
         DBX385_0 : Bool;
         DBX385_1 : Bool;
         DBX385_2 : Bool;
         DBX385_3 : Bool;
         DBX385_4 : Bool;
         DBX385_5 : Bool;
         DBX385_6 : Bool;
         DBX385_7 : Bool;
         DBX386_0 : Bool;
         DBX386_1 : Bool;   // 8;Z16 T7A Loading Unload;Eroare Generala LEV2;TK;W2;23;O
         DBX386_2 : Bool;   // 8;Z16 T7A Loading Unload;Zona Destinatie Plina;TK;W2;23;O
         DBX386_3 : Bool;   // 8;Z16 T7A Loading Unload;Zona Sursa Goala;TK;W2;23;O
         DBX386_4 : Bool;
         DBX386_5 : Bool;
         DBX386_6 : Bool;
         DBX386_7 : Bool;
         DBX387_0 : Bool;
         DBX387_1 : Bool;
         DBX387_2 : Bool;
         DBX387_3 : Bool;
         DBX387_4 : Bool;
         DBX387_5 : Bool;
         DBX387_6 : Bool;
         DBX387_7 : Bool;
         DBX388_0 : Bool;
         DBX388_1 : Bool;
         DBX388_2 : Bool;
         DBX388_3 : Bool;
         DBX388_4 : Bool;
         DBX388_5 : Bool;
         DBX388_6 : Bool;
         DBX388_7 : Bool;
         DBX389_0 : Bool;
         DBX389_1 : Bool;
         DBX389_2 : Bool;
         DBX389_3 : Bool;
         DBX389_4 : Bool;
         DBX389_5 : Bool;
         DBX389_6 : Bool;
         DBX389_7 : Bool;
         DBX390_0 : Bool;
         DBX390_1 : Bool;
         DBX390_2 : Bool;
         DBX390_3 : Bool;
         DBX390_4 : Bool;
         DBX390_5 : Bool;
         DBX390_6 : Bool;   // 8;Z17 Cool.Bench T7A Exit Check;Eroare Generala LEV2;TK;W2;23;O
         DBX390_7 : Bool;
         DBX391_0 : Bool;   // 8;Z17 Cool.Bench T7A Unload;Eroare Generala LEV2;TK;W2;23;O
         DBX391_1 : Bool;   // 8;Z17 Cool.Bench T7A Unload;Destination Zone Ful;TK;W2;23;O
         DBX391_2 : Bool;   // 8;Z17 Cool.Bench T7A Unload;Zona Sursa Goala;TK;W2;23;O
         DBX391_3 : Bool;
         DBX391_4 : Bool;
         DBX391_5 : Bool;
         DBX391_6 : Bool;
         DBX391_7 : Bool;
         DBX392_0 : Bool;
         DBX392_1 : Bool;
         DBX392_2 : Bool;
         DBX392_3 : Bool;
         DBX392_4 : Bool;
         DBX392_5 : Bool;
         DBX392_6 : Bool;
         DBX392_7 : Bool;
         DBX393_0 : Bool;
         DBX393_1 : Bool;
         DBX393_2 : Bool;
         DBX393_3 : Bool;
         DBX393_4 : Bool;
         DBX393_5 : Bool;
         DBX393_6 : Bool;
         DBX393_7 : Bool;
         DBX394_0 : Bool;
         DBX394_1 : Bool;   // 9;M9 Stamping Check Product;Eroare Generala LEV2;TK;W2;24;O
         DBX394_2 : Bool;   // 9;M9 Stamping Check Product;Lipsa ID Tracking in LEV2;TK;W2;24;O
         DBX394_3 : Bool;   // 9;M9 Stamping New Item Load;Eroare Generala LEV2;TK;W2;24;O
         DBX394_4 : Bool;   // 9;M9 Stamping New Item Load;Cheie Inactiva in LEV2;TK;W2;24;O
         DBX394_5 : Bool;   // 9;M9 Stamping New Item Load;Lot Inactiv in LEV2r;TK;W2;24;O
         DBX394_6 : Bool;   // 9;M9 Stamping New Item Load;Lipsa ID Tracking in LEV2;TK;W2;24;O
         DBX394_7 : Bool;   // 9;M9 Stamping New Item Load;ID Tracking Apartine Altui Lot;TK;W2;24;O
         DBX395_0 : Bool;   // 9;M9 Stamping New Item Load;Eroare la Creare Tracking Pass;TK;W2;24;O
         DBX395_1 : Bool;   // 9;M9 Stamping Item Count;Eroare Generala LEV2;TK;W2;24;O
         DBX395_2 : Bool;   // 9;M9 Stamping Item Count;Lipsa ID Tracking in LEV2;TK;W2;24;O
         DBX395_3 : Bool;   // 9;Z18 Exit T7A Get Pipe Attributes;Eroare Generala LEV2;TK;W2;23;O
         DBX395_4 : Bool;   // 9;Z18 Exit T7A Get Pipe Attributes;Zona Destinatie Plina;TK;W2;23;O
         DBX395_5 : Bool;   // 9;Z18 Exit T7A Get Pipe Attributes;Zona Sursa Goala;TK;W2;23;O
         DBX395_6 : Bool;   // 9;Z18 Exit T7A;Role T7-A Incoerenta Tracking;TK;W2;23;O
         DBX395_7 : Bool;
         DBX396_0 : Bool;
         DBX396_1 : Bool;   // 9;Send Data Stamping Machine;Eroare Generala LEV2;TK;W2;24;O
         DBX396_2 : Bool;   // 9;Send Data Stamping Machine;Lipsa ID Tracking in LEV2;TK;W2;24;O
         DBX396_3 : Bool;   // 9;Send Data Stamping Machine;Lipsa Mesaj Marcare;TK;W2;24;O
         DBX396_4 : Bool;   // 9;Send Data Stamping Machine;Masina Marcare Eroare Comunicatie;TK;W2;24;O
         DBX396_5 : Bool;   // 9;Send Data Stamping Machine;Tip Mesaj Marcare Invalid;TK;W2;24;O
         DBX396_6 : Bool;
         DBX396_7 : Bool;
         DBX397_0 : Bool;
         DBX397_1 : Bool;   // 9;Send Data Stamping Machine Robot;Eroare Generala LEV2;TK;W2;24;O
         DBX397_2 : Bool;   // 9;Send Data Stamping Machine Robot;Lipsa ID Tracking in LEV2;TK;W2;24;O
         DBX397_3 : Bool;   // 9;Send Data Stamping Machine Robot;Lipsa Mesaj Marcare;TK;W2;24;O
         DBX397_4 : Bool;   // 9;Send Data Stamping Machine Robo;Masina Marcare Eroare Comunicatie;TK;W2;24;O
         DBX397_5 : Bool;   // 9;Send Data Stamping Machine Robot;Tip Mesaj Marcare Invalid;TK;W2;24;O
         DBX397_6 : Bool;
         DBX397_7 : Bool;
         DBX398_0 : Bool;
         DBX398_1 : Bool;
         DBX398_2 : Bool;
         DBX398_3 : Bool;
         DBX398_4 : Bool;
         DBX398_5 : Bool;
         DBX398_6 : Bool;
         DBX398_7 : Bool;
         DBX399_0 : Bool;
         DBX399_1 : Bool;
         DBX399_2 : Bool;
         DBX399_3 : Bool;
         DBX399_4 : Bool;
         DBX399_5 : Bool;
         DBX399_6 : Bool;
         DBX399_7 : Bool;
      END_STRUCT;
      TAB_02 : Struct
         CNT02 : Int;
         DBX402_0 : Bool;
         DBX402_1 : Bool;
         DBX402_2 : Bool;
         DBX402_3 : Bool;
         DBX402_4 : Bool;
         DBX402_5 : Bool;
         DBX402_6 : Bool;
         DBX402_7 : Bool;
         DBX403_0 : Bool;
         DBX403_1 : Bool;
         DBX403_2 : Bool;
         DBX403_3 : Bool;
         DBX403_4 : Bool;
         DBX403_5 : Bool;
         DBX403_6 : Bool;
         DBX403_7 : Bool;
         DBX404_0 : Bool;
         DBX404_1 : Bool;
         DBX404_2 : Bool;
         DBX404_3 : Bool;
         DBX404_4 : Bool;
         DBX404_5 : Bool;
         DBX404_6 : Bool;
         DBX404_7 : Bool;
         DBX405_0 : Bool;
         DBX405_1 : Bool;
         DBX405_2 : Bool;
         DBX405_3 : Bool;
         DBX405_4 : Bool;
         DBX405_5 : Bool;
         DBX405_6 : Bool;
         DBX405_7 : Bool;
         DBX406_0 : Bool;
         DBX406_1 : Bool;
         DBX406_2 : Bool;
         DBX406_3 : Bool;
         DBX406_4 : Bool;
         DBX406_5 : Bool;
         DBX406_6 : Bool;
         DBX406_7 : Bool;
         DBX407_0 : Bool;
         DBX407_1 : Bool;
         DBX407_2 : Bool;
         DBX407_3 : Bool;
         DBX407_4 : Bool;
         DBX407_5 : Bool;
         DBX407_6 : Bool;
         DBX407_7 : Bool;
         DBX408_0 : Bool;
         DBX408_1 : Bool;
         DBX408_2 : Bool;
         DBX408_3 : Bool;
         DBX408_4 : Bool;
         DBX408_5 : Bool;
         DBX408_6 : Bool;
         DBX408_7 : Bool;
         DBX409_0 : Bool;
         DBX409_1 : Bool;
         DBX409_2 : Bool;
         DBX409_3 : Bool;
         DBX409_4 : Bool;
         DBX409_5 : Bool;
         DBX409_6 : Bool;
         DBX409_7 : Bool;
         DBX410_0 : Bool;
         DBX410_1 : Bool;
         DBX410_2 : Bool;
         DBX410_3 : Bool;
         DBX410_4 : Bool;
         DBX410_5 : Bool;
         DBX410_6 : Bool;
         DBX410_7 : Bool;
         DBX411_0 : Bool;
         DBX411_1 : Bool;
         DBX411_2 : Bool;
         DBX411_3 : Bool;
         DBX411_4 : Bool;
         DBX411_5 : Bool;
         DBX411_6 : Bool;
         DBX411_7 : Bool;
         DBX412_0 : Bool;
         DBX412_1 : Bool;
         DBX412_2 : Bool;
         DBX412_3 : Bool;
         DBX412_4 : Bool;
         DBX412_5 : Bool;
         DBX412_6 : Bool;
         DBX412_7 : Bool;
         DBX413_0 : Bool;
         DBX413_1 : Bool;
         DBX413_2 : Bool;
         DBX413_3 : Bool;
         DBX413_4 : Bool;
         DBX413_5 : Bool;
         DBX413_6 : Bool;
         DBX413_7 : Bool;
         DBX414_0 : Bool;
         DBX414_1 : Bool;
         DBX414_2 : Bool;
         DBX414_3 : Bool;
         DBX414_4 : Bool;
         DBX414_5 : Bool;
         DBX414_6 : Bool;
         DBX414_7 : Bool;
         DBX415_0 : Bool;
         DBX415_1 : Bool;
         DBX415_2 : Bool;
         DBX415_3 : Bool;
         DBX415_4 : Bool;
         DBX415_5 : Bool;
         DBX415_6 : Bool;
         DBX415_7 : Bool;
         DBX416_0 : Bool;
         DBX416_1 : Bool;
         DBX416_2 : Bool;
         DBX416_3 : Bool;
         DBX416_4 : Bool;
         DBX416_5 : Bool;
         DBX416_6 : Bool;
         DBX416_7 : Bool;
         DBX417_0 : Bool;
         DBX417_1 : Bool;
         DBX417_2 : Bool;
         DBX417_3 : Bool;
         DBX417_4 : Bool;
         DBX417_5 : Bool;
         DBX417_6 : Bool;
         DBX417_7 : Bool;
         DBX418_0 : Bool;
         DBX418_1 : Bool;
         DBX418_2 : Bool;
         DBX418_3 : Bool;
         DBX418_4 : Bool;
         DBX418_5 : Bool;
         DBX418_6 : Bool;
         DBX418_7 : Bool;
         DBX419_0 : Bool;
         DBX419_1 : Bool;
         DBX419_2 : Bool;
         DBX419_3 : Bool;
         DBX419_4 : Bool;
         DBX419_5 : Bool;
         DBX419_6 : Bool;
         DBX419_7 : Bool;
         DBX420_0 : Bool;
         DBX420_1 : Bool;
         DBX420_2 : Bool;
         DBX420_3 : Bool;
         DBX420_4 : Bool;
         DBX420_5 : Bool;
         DBX420_6 : Bool;
         DBX420_7 : Bool;
         DBX421_0 : Bool;
         DBX421_1 : Bool;
         DBX421_2 : Bool;
         DBX421_3 : Bool;
         DBX421_4 : Bool;
         DBX421_5 : Bool;
         DBX421_6 : Bool;
         DBX421_7 : Bool;
         DBX422_0 : Bool;
         DBX422_1 : Bool;
         DBX422_2 : Bool;
         DBX422_3 : Bool;
         DBX422_4 : Bool;
         DBX422_5 : Bool;
         DBX422_6 : Bool;
         DBX422_7 : Bool;
         DBX423_0 : Bool;
         DBX423_1 : Bool;
         DBX423_2 : Bool;
         DBX423_3 : Bool;
         DBX423_4 : Bool;
         DBX423_5 : Bool;
         DBX423_6 : Bool;
         DBX423_7 : Bool;
         DBX424_0 : Bool;
         DBX424_1 : Bool;
         DBX424_2 : Bool;
         DBX424_3 : Bool;
         DBX424_4 : Bool;
         DBX424_5 : Bool;
         DBX424_6 : Bool;
         DBX424_7 : Bool;
         DBX425_0 : Bool;
         DBX425_1 : Bool;
         DBX425_2 : Bool;
         DBX425_3 : Bool;
         DBX425_4 : Bool;
         DBX425_5 : Bool;
         DBX425_6 : Bool;
         DBX425_7 : Bool;
         DBX426_0 : Bool;
         DBX426_1 : Bool;
         DBX426_2 : Bool;
         DBX426_3 : Bool;
         DBX426_4 : Bool;
         DBX426_5 : Bool;
         DBX426_6 : Bool;
         DBX426_7 : Bool;
         DBX427_0 : Bool;
         DBX427_1 : Bool;
         DBX427_2 : Bool;
         DBX427_3 : Bool;
         DBX427_4 : Bool;
         DBX427_5 : Bool;
         DBX427_6 : Bool;
         DBX427_7 : Bool;
         DBX428_0 : Bool;
         DBX428_1 : Bool;
         DBX428_2 : Bool;
         DBX428_3 : Bool;
         DBX428_4 : Bool;
         DBX428_5 : Bool;
         DBX428_6 : Bool;
         DBX428_7 : Bool;
         DBX429_0 : Bool;
         DBX429_1 : Bool;
         DBX429_2 : Bool;
         DBX429_3 : Bool;
         DBX429_4 : Bool;
         DBX429_5 : Bool;
         DBX429_6 : Bool;
         DBX429_7 : Bool;
         DBX430_0 : Bool;
         DBX430_1 : Bool;
         DBX430_2 : Bool;
         DBX430_3 : Bool;
         DBX430_4 : Bool;
         DBX430_5 : Bool;
         DBX430_6 : Bool;
         DBX430_7 : Bool;
         DBX431_0 : Bool;
         DBX431_1 : Bool;
         DBX431_2 : Bool;
         DBX431_3 : Bool;
         DBX431_4 : Bool;
         DBX431_5 : Bool;
         DBX431_6 : Bool;
         DBX431_7 : Bool;
         DBX432_0 : Bool;
         DBX432_1 : Bool;
         DBX432_2 : Bool;
         DBX432_3 : Bool;
         DBX432_4 : Bool;
         DBX432_5 : Bool;
         DBX432_6 : Bool;
         DBX432_7 : Bool;
         DBX433_0 : Bool;
         DBX433_1 : Bool;
         DBX433_2 : Bool;
         DBX433_3 : Bool;
         DBX433_4 : Bool;
         DBX433_5 : Bool;
         DBX433_6 : Bool;
         DBX433_7 : Bool;
         DBX434_0 : Bool;
         DBX434_1 : Bool;
         DBX434_2 : Bool;
         DBX434_3 : Bool;
         DBX434_4 : Bool;
         DBX434_5 : Bool;
         DBX434_6 : Bool;
         DBX434_7 : Bool;
         DBX435_0 : Bool;
         DBX435_1 : Bool;
         DBX435_2 : Bool;
         DBX435_3 : Bool;
         DBX435_4 : Bool;
         DBX435_5 : Bool;
         DBX435_6 : Bool;
         DBX435_7 : Bool;
         DBX436_0 : Bool;
         DBX436_1 : Bool;
         DBX436_2 : Bool;
         DBX436_3 : Bool;
         DBX436_4 : Bool;
         DBX436_5 : Bool;
         DBX436_6 : Bool;
         DBX436_7 : Bool;
         DBX437_0 : Bool;
         DBX437_1 : Bool;
         DBX437_2 : Bool;
         DBX437_3 : Bool;
         DBX437_4 : Bool;
         DBX437_5 : Bool;
         DBX437_6 : Bool;
         DBX437_7 : Bool;
         DBX438_0 : Bool;
         DBX438_1 : Bool;
         DBX438_2 : Bool;
         DBX438_3 : Bool;
         DBX438_4 : Bool;
         DBX438_5 : Bool;
         DBX438_6 : Bool;
         DBX438_7 : Bool;
         DBX439_0 : Bool;
         DBX439_1 : Bool;
         DBX439_2 : Bool;
         DBX439_3 : Bool;
         DBX439_4 : Bool;
         DBX439_5 : Bool;
         DBX439_6 : Bool;
         DBX439_7 : Bool;
         DBX440_0 : Bool;
         DBX440_1 : Bool;
         DBX440_2 : Bool;
         DBX440_3 : Bool;
         DBX440_4 : Bool;
         DBX440_5 : Bool;
         DBX440_6 : Bool;
         DBX440_7 : Bool;
         DBX441_0 : Bool;
         DBX441_1 : Bool;
         DBX441_2 : Bool;
         DBX441_3 : Bool;
         DBX441_4 : Bool;
         DBX441_5 : Bool;
         DBX441_6 : Bool;
         DBX441_7 : Bool;
         DBX442_0 : Bool;
         DBX442_1 : Bool;
         DBX442_2 : Bool;
         DBX442_3 : Bool;
         DBX442_4 : Bool;
         DBX442_5 : Bool;
         DBX442_6 : Bool;
         DBX442_7 : Bool;
         DBX443_0 : Bool;
         DBX443_1 : Bool;
         DBX443_2 : Bool;
         DBX443_3 : Bool;
         DBX443_4 : Bool;
         DBX443_5 : Bool;
         DBX443_6 : Bool;
         DBX443_7 : Bool;
         DBX444_0 : Bool;
         DBX444_1 : Bool;
         DBX444_2 : Bool;
         DBX444_3 : Bool;
         DBX444_4 : Bool;
         DBX444_5 : Bool;
         DBX444_6 : Bool;
         DBX444_7 : Bool;
         DBX445_0 : Bool;
         DBX445_1 : Bool;
         DBX445_2 : Bool;
         DBX445_3 : Bool;
         DBX445_4 : Bool;
         DBX445_5 : Bool;
         DBX445_6 : Bool;
         DBX445_7 : Bool;
         DBX446_0 : Bool;
         DBX446_1 : Bool;
         DBX446_2 : Bool;
         DBX446_3 : Bool;
         DBX446_4 : Bool;
         DBX446_5 : Bool;
         DBX446_6 : Bool;
         DBX446_7 : Bool;
         DBX447_0 : Bool;
         DBX447_1 : Bool;
         DBX447_2 : Bool;
         DBX447_3 : Bool;
         DBX447_4 : Bool;
         DBX447_5 : Bool;
         DBX447_6 : Bool;
         DBX447_7 : Bool;
         DBX448_0 : Bool;
         DBX448_1 : Bool;
         DBX448_2 : Bool;
         DBX448_3 : Bool;
         DBX448_4 : Bool;
         DBX448_5 : Bool;
         DBX448_6 : Bool;
         DBX448_7 : Bool;
         DBX449_0 : Bool;
         DBX449_1 : Bool;
         DBX449_2 : Bool;
         DBX449_3 : Bool;
         DBX449_4 : Bool;
         DBX449_5 : Bool;
         DBX449_6 : Bool;
         DBX449_7 : Bool;
         DBX450_0 : Bool;
         DBX450_1 : Bool;
         DBX450_2 : Bool;
         DBX450_3 : Bool;
         DBX450_4 : Bool;
         DBX450_5 : Bool;
         DBX450_6 : Bool;
         DBX450_7 : Bool;
         DBX451_0 : Bool;
         DBX451_1 : Bool;
         DBX451_2 : Bool;
         DBX451_3 : Bool;
         DBX451_4 : Bool;
         DBX451_5 : Bool;
         DBX451_6 : Bool;
         DBX451_7 : Bool;
         DBX452_0 : Bool;
         DBX452_1 : Bool;
         DBX452_2 : Bool;
         DBX452_3 : Bool;
         DBX452_4 : Bool;
         DBX452_5 : Bool;
         DBX452_6 : Bool;
         DBX452_7 : Bool;
         DBX453_0 : Bool;
         DBX453_1 : Bool;
         DBX453_2 : Bool;
         DBX453_3 : Bool;
         DBX453_4 : Bool;
         DBX453_5 : Bool;
         DBX453_6 : Bool;
         DBX453_7 : Bool;
         DBX454_0 : Bool;
         DBX454_1 : Bool;
         DBX454_2 : Bool;
         DBX454_3 : Bool;
         DBX454_4 : Bool;
         DBX454_5 : Bool;
         DBX454_6 : Bool;
         DBX454_7 : Bool;
         DBX455_0 : Bool;
         DBX455_1 : Bool;
         DBX455_2 : Bool;
         DBX455_3 : Bool;
         DBX455_4 : Bool;
         DBX455_5 : Bool;
         DBX455_6 : Bool;
         DBX455_7 : Bool;
         DBX456_0 : Bool;
         DBX456_1 : Bool;
         DBX456_2 : Bool;
         DBX456_3 : Bool;
         DBX456_4 : Bool;
         DBX456_5 : Bool;
         DBX456_6 : Bool;
         DBX456_7 : Bool;
         DBX457_0 : Bool;
         DBX457_1 : Bool;
         DBX457_2 : Bool;
         DBX457_3 : Bool;
         DBX457_4 : Bool;
         DBX457_5 : Bool;
         DBX457_6 : Bool;
         DBX457_7 : Bool;
         DBX458_0 : Bool;
         DBX458_1 : Bool;
         DBX458_2 : Bool;
         DBX458_3 : Bool;
         DBX458_4 : Bool;
         DBX458_5 : Bool;
         DBX458_6 : Bool;
         DBX458_7 : Bool;
         DBX459_0 : Bool;
         DBX459_1 : Bool;
         DBX459_2 : Bool;
         DBX459_3 : Bool;
         DBX459_4 : Bool;
         DBX459_5 : Bool;
         DBX459_6 : Bool;
         DBX459_7 : Bool;
         DBX460_0 : Bool;
         DBX460_1 : Bool;
         DBX460_2 : Bool;
         DBX460_3 : Bool;
         DBX460_4 : Bool;
         DBX460_5 : Bool;
         DBX460_6 : Bool;
         DBX460_7 : Bool;
         DBX461_0 : Bool;
         DBX461_1 : Bool;
         DBX461_2 : Bool;
         DBX461_3 : Bool;
         DBX461_4 : Bool;
         DBX461_5 : Bool;
         DBX461_6 : Bool;
         DBX461_7 : Bool;
         DBX462_0 : Bool;
         DBX462_1 : Bool;
         DBX462_2 : Bool;
         DBX462_3 : Bool;
         DBX462_4 : Bool;
         DBX462_5 : Bool;
         DBX462_6 : Bool;
         DBX462_7 : Bool;
         DBX463_0 : Bool;
         DBX463_1 : Bool;
         DBX463_2 : Bool;
         DBX463_3 : Bool;
         DBX463_4 : Bool;
         DBX463_5 : Bool;
         DBX463_6 : Bool;
         DBX463_7 : Bool;
         DBX464_0 : Bool;
         DBX464_1 : Bool;
         DBX464_2 : Bool;
         DBX464_3 : Bool;
         DBX464_4 : Bool;
         DBX464_5 : Bool;
         DBX464_6 : Bool;
         DBX464_7 : Bool;
         DBX465_0 : Bool;
         DBX465_1 : Bool;
         DBX465_2 : Bool;
         DBX465_3 : Bool;
         DBX465_4 : Bool;
         DBX465_5 : Bool;
         DBX465_6 : Bool;
         DBX465_7 : Bool;
         DBX466_0 : Bool;
         DBX466_1 : Bool;
         DBX466_2 : Bool;
         DBX466_3 : Bool;
         DBX466_4 : Bool;
         DBX466_5 : Bool;
         DBX466_6 : Bool;
         DBX466_7 : Bool;
         DBX467_0 : Bool;
         DBX467_1 : Bool;
         DBX467_2 : Bool;
         DBX467_3 : Bool;
         DBX467_4 : Bool;
         DBX467_5 : Bool;
         DBX467_6 : Bool;
         DBX467_7 : Bool;
         DBX468_0 : Bool;
         DBX468_1 : Bool;
         DBX468_2 : Bool;
         DBX468_3 : Bool;
         DBX468_4 : Bool;
         DBX468_5 : Bool;
         DBX468_6 : Bool;
         DBX468_7 : Bool;
         DBX469_0 : Bool;
         DBX469_1 : Bool;
         DBX469_2 : Bool;
         DBX469_3 : Bool;
         DBX469_4 : Bool;
         DBX469_5 : Bool;
         DBX469_6 : Bool;
         DBX469_7 : Bool;
         DBX470_0 : Bool;
         DBX470_1 : Bool;
         DBX470_2 : Bool;
         DBX470_3 : Bool;
         DBX470_4 : Bool;
         DBX470_5 : Bool;
         DBX470_6 : Bool;
         DBX470_7 : Bool;
         DBX471_0 : Bool;
         DBX471_1 : Bool;
         DBX471_2 : Bool;
         DBX471_3 : Bool;
         DBX471_4 : Bool;
         DBX471_5 : Bool;
         DBX471_6 : Bool;
         DBX471_7 : Bool;
         DBX472_0 : Bool;
         DBX472_1 : Bool;
         DBX472_2 : Bool;
         DBX472_3 : Bool;
         DBX472_4 : Bool;
         DBX472_5 : Bool;
         DBX472_6 : Bool;
         DBX472_7 : Bool;
         DBX473_0 : Bool;
         DBX473_1 : Bool;
         DBX473_2 : Bool;
         DBX473_3 : Bool;
         DBX473_4 : Bool;
         DBX473_5 : Bool;
         DBX473_6 : Bool;
         DBX473_7 : Bool;
         DBX474_0 : Bool;
         DBX474_1 : Bool;
         DBX474_2 : Bool;
         DBX474_3 : Bool;
         DBX474_4 : Bool;
         DBX474_5 : Bool;
         DBX474_6 : Bool;
         DBX474_7 : Bool;
         DBX475_0 : Bool;
         DBX475_1 : Bool;
         DBX475_2 : Bool;
         DBX475_3 : Bool;
         DBX475_4 : Bool;
         DBX475_5 : Bool;
         DBX475_6 : Bool;
         DBX475_7 : Bool;
         DBX476_0 : Bool;
         DBX476_1 : Bool;
         DBX476_2 : Bool;
         DBX476_3 : Bool;
         DBX476_4 : Bool;
         DBX476_5 : Bool;
         DBX476_6 : Bool;
         DBX476_7 : Bool;
         DBX477_0 : Bool;
         DBX477_1 : Bool;
         DBX477_2 : Bool;
         DBX477_3 : Bool;
         DBX477_4 : Bool;
         DBX477_5 : Bool;
         DBX477_6 : Bool;
         DBX477_7 : Bool;
         DBX478_0 : Bool;
         DBX478_1 : Bool;
         DBX478_2 : Bool;
         DBX478_3 : Bool;
         DBX478_4 : Bool;
         DBX478_5 : Bool;
         DBX478_6 : Bool;
         DBX478_7 : Bool;
         DBX479_0 : Bool;
         DBX479_1 : Bool;
         DBX479_2 : Bool;
         DBX479_3 : Bool;
         DBX479_4 : Bool;
         DBX479_5 : Bool;
         DBX479_6 : Bool;
         DBX479_7 : Bool;
         DBX480_0 : Bool;
         DBX480_1 : Bool;
         DBX480_2 : Bool;
         DBX480_3 : Bool;
         DBX480_4 : Bool;
         DBX480_5 : Bool;
         DBX480_6 : Bool;
         DBX480_7 : Bool;
         DBX481_0 : Bool;
         DBX481_1 : Bool;
         DBX481_2 : Bool;
         DBX481_3 : Bool;
         DBX481_4 : Bool;
         DBX481_5 : Bool;
         DBX481_6 : Bool;
         DBX481_7 : Bool;
         DBX482_0 : Bool;
         DBX482_1 : Bool;
         DBX482_2 : Bool;
         DBX482_3 : Bool;
         DBX482_4 : Bool;
         DBX482_5 : Bool;
         DBX482_6 : Bool;
         DBX482_7 : Bool;
         DBX483_0 : Bool;
         DBX483_1 : Bool;
         DBX483_2 : Bool;
         DBX483_3 : Bool;
         DBX483_4 : Bool;
         DBX483_5 : Bool;
         DBX483_6 : Bool;
         DBX483_7 : Bool;
         DBX484_0 : Bool;
         DBX484_1 : Bool;
         DBX484_2 : Bool;
         DBX484_3 : Bool;
         DBX484_4 : Bool;
         DBX484_5 : Bool;
         DBX484_6 : Bool;
         DBX484_7 : Bool;
         DBX485_0 : Bool;
         DBX485_1 : Bool;
         DBX485_2 : Bool;
         DBX485_3 : Bool;
         DBX485_4 : Bool;
         DBX485_5 : Bool;
         DBX485_6 : Bool;
         DBX485_7 : Bool;
         DBX486_0 : Bool;
         DBX486_1 : Bool;
         DBX486_2 : Bool;
         DBX486_3 : Bool;
         DBX486_4 : Bool;
         DBX486_5 : Bool;
         DBX486_6 : Bool;
         DBX486_7 : Bool;
         DBX487_0 : Bool;
         DBX487_1 : Bool;
         DBX487_2 : Bool;
         DBX487_3 : Bool;
         DBX487_4 : Bool;
         DBX487_5 : Bool;
         DBX487_6 : Bool;
         DBX487_7 : Bool;
         DBX488_0 : Bool;
         DBX488_1 : Bool;
         DBX488_2 : Bool;
         DBX488_3 : Bool;
         DBX488_4 : Bool;
         DBX488_5 : Bool;
         DBX488_6 : Bool;
         DBX488_7 : Bool;
         DBX489_0 : Bool;
         DBX489_1 : Bool;
         DBX489_2 : Bool;
         DBX489_3 : Bool;
         DBX489_4 : Bool;
         DBX489_5 : Bool;
         DBX489_6 : Bool;
         DBX489_7 : Bool;
         DBX490_0 : Bool;
         DBX490_1 : Bool;
         DBX490_2 : Bool;
         DBX490_3 : Bool;
         DBX490_4 : Bool;
         DBX490_5 : Bool;
         DBX490_6 : Bool;
         DBX490_7 : Bool;
         DBX491_0 : Bool;
         DBX491_1 : Bool;
         DBX491_2 : Bool;
         DBX491_3 : Bool;
         DBX491_4 : Bool;
         DBX491_5 : Bool;
         DBX491_6 : Bool;
         DBX491_7 : Bool;
         DBX492_0 : Bool;
         DBX492_1 : Bool;
         DBX492_2 : Bool;
         DBX492_3 : Bool;
         DBX492_4 : Bool;
         DBX492_5 : Bool;
         DBX492_6 : Bool;
         DBX492_7 : Bool;
         DBX493_0 : Bool;
         DBX493_1 : Bool;
         DBX493_2 : Bool;
         DBX493_3 : Bool;
         DBX493_4 : Bool;
         DBX493_5 : Bool;
         DBX493_6 : Bool;
         DBX493_7 : Bool;
         DBX494_0 : Bool;
         DBX494_1 : Bool;
         DBX494_2 : Bool;
         DBX494_3 : Bool;
         DBX494_4 : Bool;
         DBX494_5 : Bool;
         DBX494_6 : Bool;
         DBX494_7 : Bool;
         DBX495_0 : Bool;
         DBX495_1 : Bool;
         DBX495_2 : Bool;
         DBX495_3 : Bool;
         DBX495_4 : Bool;
         DBX495_5 : Bool;
         DBX495_6 : Bool;
         DBX495_7 : Bool;
         DBX496_0 : Bool;
         DBX496_1 : Bool;
         DBX496_2 : Bool;
         DBX496_3 : Bool;
         DBX496_4 : Bool;
         DBX496_5 : Bool;
         DBX496_6 : Bool;
         DBX496_7 : Bool;
         DBX497_0 : Bool;
         DBX497_1 : Bool;
         DBX497_2 : Bool;
         DBX497_3 : Bool;
         DBX497_4 : Bool;
         DBX497_5 : Bool;
         DBX497_6 : Bool;
         DBX497_7 : Bool;
         DBX498_0 : Bool;
         DBX498_1 : Bool;
         DBX498_2 : Bool;
         DBX498_3 : Bool;
         DBX498_4 : Bool;
         DBX498_5 : Bool;
         DBX498_6 : Bool;
         DBX498_7 : Bool;
         DBX499_0 : Bool;
         DBX499_1 : Bool;
         DBX499_2 : Bool;
         DBX499_3 : Bool;
         DBX499_4 : Bool;
         DBX499_5 : Bool;
         DBX499_6 : Bool;
         DBX499_7 : Bool;
         DBX500_0 : Bool;
         DBX500_1 : Bool;
         DBX500_2 : Bool;
         DBX500_3 : Bool;
         DBX500_4 : Bool;
         DBX500_5 : Bool;
         DBX500_6 : Bool;
         DBX500_7 : Bool;
         DBX501_0 : Bool;   // 1;LEV2;HSK01-DPL.LD.CREATE-Recoverable error;TK;W0;N;O;M
         DBX501_1 : Bool;   // 1;LEV2;HSK01-DPL.LD.CREATE-Error;TK;W0;N;O;M
         DBX501_2 : Bool;   // 1;LEV2;HSK01-DPL.LD.CREATE-Time out error;TK;W0;N;O;M
         DBX501_3 : Bool;   // 1;LEV2;HSK01-DPL.LD.CREATE-Configuration error;TK;W0;N;O;M
         DBX501_4 : Bool;   // 1;LEV2;HSK01-DPL.LD.CREATE-Lock;TK;W0;N;O;M
         DBX501_5 : Bool;
         DBX501_6 : Bool;
         DBX501_7 : Bool;
         DBX502_0 : Bool;   // 1;LEV2;HSK02-DPL.LD.COUNT-Recoverable error;TK;W0;N;O;M
         DBX502_1 : Bool;   // 1;LEV2;HSK02-DPL.LD.COUNT-Error;TK;W0;N;O;M
         DBX502_2 : Bool;   // 1;LEV2;HSK02-DPL.LD.COUNT-Time out error;TK;W0;N;O;M
         DBX502_3 : Bool;   // 1;LEV2;HSK02-DPL.LD.COUNT-Configuration error;TK;W0;N;O;M
         DBX502_4 : Bool;   // 1;LEV2;HSK02-DPL.LD.COUNT-Lock;TK;W0;N;O;M
         DBX502_5 : Bool;
         DBX502_6 : Bool;
         DBX502_7 : Bool;
         DBX503_0 : Bool;   // 1;LEV2;HSK03-DPL.R1.MOVE-Recoverable error;TK;W0;N;O;M
         DBX503_1 : Bool;   // 1;LEV2;HSK03-DPL.R1.MOVE-Error;TK;W0;N;O;M
         DBX503_2 : Bool;   // 1;LEV2;HSK03-DPL.R1.MOVE-Time out error;TK;W0;N;O;M
         DBX503_3 : Bool;   // 1;LEV2;HSK03-DPL.R1.MOVE-Configuration error;TK;W0;N;O;M
         DBX503_4 : Bool;   // 1;LEV2;HSK03-DPL.R1.MOVE-Lock;TK;W0;N;O;M
         DBX503_5 : Bool;
         DBX503_6 : Bool;
         DBX503_7 : Bool;
         DBX504_0 : Bool;   // 1;LEV2;HSK04-DPL.R2.MOVE-Recoverable error;TK;W0;N;O;M
         DBX504_1 : Bool;   // 1;LEV2;HSK04-DPL.R2.MOVE-Error;TK;W0;N;O;M
         DBX504_2 : Bool;   // 1;LEV2;HSK04-DPL.R2.MOVE-Time out error;TK;W0;N;O;M
         DBX504_3 : Bool;   // 1;LEV2;HSK04-DPL.R2.MOVE-Configuration error;TK;W0;N;O;M
         DBX504_4 : Bool;   // 1;LEV2;HSK04-DPL.R2.MOVE-Lock;TK;W0;N;O;M
         DBX504_5 : Bool;
         DBX504_6 : Bool;
         DBX504_7 : Bool;
         DBX505_0 : Bool;   // 1;LEV2;HSK05-DPL.WSH.BEGIN-Recoverable error;TK;W0;N;O;M
         DBX505_1 : Bool;   // 1;LEV2;HSK05-DPL.WSH.BEGIN-Error;TK;W0;N;O;M
         DBX505_2 : Bool;   // 1;LEV2;HSK05-DPL.WSH.BEGIN-Time out error;TK;W0;N;O;M
         DBX505_3 : Bool;   // 1;LEV2;HSK05-DPL.WSH.BEGIN-Configuration error;TK;W0;N;O;M
         DBX505_4 : Bool;   // 1;LEV2;HSK05-DPL.WSH.BEGIN-Lock;TK;W0;N;O;M
         DBX505_5 : Bool;
         DBX505_6 : Bool;
         DBX505_7 : Bool;
         DBX506_0 : Bool;   // 1;LEV2;HSK06-DPL.WSH.END-Recoverable error;TK;W0;N;O;M
         DBX506_1 : Bool;   // 1;LEV2;HSK06-DPL.WSH.END-Error;TK;W0;N;O;M
         DBX506_2 : Bool;   // 1;LEV2;HSK06-DPL.WSH.END-Time out error;TK;W0;N;O;M
         DBX506_3 : Bool;   // 1;LEV2;HSK06-DPL.WSH.END-Configuration error;TK;W0;N;O;M
         DBX506_4 : Bool;   // 1;LEV2;HSK06-DPL.WSH.END-Lock;TK;W0;N;O;M
         DBX506_5 : Bool;
         DBX506_6 : Bool;
         DBX506_7 : Bool;
         DBX507_0 : Bool;   // 1;LEV2;HSK07-DPL.PREH.BEGIN-Recoverable error;TK;W0;N;O;M
         DBX507_1 : Bool;   // 1;LEV2;HSK07-DPL.PREH.BEGIN-Error;TK;W0;N;O;M
         DBX507_2 : Bool;   // 1;LEV2;HSK07-DPL.PREH.BEGIN-Time out error;TK;W0;N;O;M
         DBX507_3 : Bool;   // 1;LEV2;HSK07-DPL.PREH.BEGIN-Configuration error;TK;W0;N;O;M
         DBX507_4 : Bool;   // 1;LEV2;HSK07-DPL.PREH.BEGIN-Lock;TK;W0;N;O;M
         DBX507_5 : Bool;
         DBX507_6 : Bool;
         DBX507_7 : Bool;
         DBX508_0 : Bool;   // 1;LEV2;HSK08-DPL.PREH.END-Recoverable error;TK;W0;N;O;M
         DBX508_1 : Bool;   // 1;LEV2;HSK08-DPL.PREH.END-Error;TK;W0;N;O;M
         DBX508_2 : Bool;   // 1;LEV2;HSK08-DPL.PREH.END-Time out error;TK;W0;N;O;M
         DBX508_3 : Bool;   // 1;LEV2;HSK08-DPL.PREH.END-Configuration error;TK;W0;N;O;M
         DBX508_4 : Bool;   // 1;LEV2;HSK08-DPL.PREH.END-Lock;TK;W0;N;O;M
         DBX508_5 : Bool;
         DBX508_6 : Bool;
         DBX508_7 : Bool;
         DBX509_0 : Bool;   // 1;LEV2;HSK09-DPL.COA.BEGIN-Recoverable error;TK;W0;N;O;M
         DBX509_1 : Bool;   // 1;LEV2;HSK09-DPL.COA.BEGIN-Error;TK;W0;N;O;M
         DBX509_2 : Bool;   // 1;LEV2;HSK09-DPL.COA.BEGIN-Time out error;TK;W0;N;O;M
         DBX509_3 : Bool;   // 1;LEV2;HSK09-DPL.COA.BEGIN-Configuration error;TK;W0;N;O;M
         DBX509_4 : Bool;   // 1;LEV2;HSK09-DPL.COA.BEGIN-Lock;TK;W0;N;O;M
         DBX509_5 : Bool;
         DBX509_6 : Bool;
         DBX509_7 : Bool;
         DBX510_0 : Bool;   // 1;LEV2;HSK10-DPL.COA.END-Recoverable error;TK;W0;N;O;M
         DBX510_1 : Bool;   // 1;LEV2;HSK10-DPL.COA.END-Error;TK;W0;N;O;M
         DBX510_2 : Bool;   // 1;LEV2;HSK10-DPL.COA.END-Time out error;TK;W0;N;O;M
         DBX510_3 : Bool;   // 1;LEV2;HSK10-DPL.COA.END-Configuration error;TK;W0;N;O;M
         DBX510_4 : Bool;   // 1;LEV2;HSK10-DPL.COA.END-Lock;TK;W0;N;O;M
         DBX510_5 : Bool;
         DBX510_6 : Bool;
         DBX510_7 : Bool;
         DBX511_0 : Bool;   // 1;LEV2;HSK11-DPL.CNG.BEGIN-Recoverable error;TK;W0;N;O;M
         DBX511_1 : Bool;   // 1;LEV2;HSK11-DPL.CNG.BEGIN-Error;TK;W0;N;O;M
         DBX511_2 : Bool;   // 1;LEV2;HSK11-DPL.CNG.BEGIN-Time out error;TK;W0;N;O;M
         DBX511_3 : Bool;   // 1;LEV2;HSK11-DPL.CNG.BEGIN-Configuration error;TK;W0;N;O;M
         DBX511_4 : Bool;   // 1;LEV2;HSK11-DPL.CNG.BEGIN-Lock;TK;W0;N;O;M
         DBX511_5 : Bool;
         DBX511_6 : Bool;
         DBX511_7 : Bool;
         DBX512_0 : Bool;   // 1;LEV2;HSK12-DPL.CNG.CHECK1-Recoverable error;TK;W0;N;O;M
         DBX512_1 : Bool;   // 1;LEV2;HSK12-DPL.CNG.CHECK1-Error;TK;W0;N;O;M
         DBX512_2 : Bool;   // 1;LEV2;HSK12-DPL.CNG.CHECK1-Time out error;TK;W0;N;O;M
         DBX512_3 : Bool;   // 1;LEV2;HSK12-DPL.CNG.CHECK1-Configuration error;TK;W0;N;O;M
         DBX512_4 : Bool;   // 1;LEV2;HSK12-DPL.CNG.CHECK1-Lock;TK;W0;N;O;M
         DBX512_5 : Bool;
         DBX512_6 : Bool;
         DBX512_7 : Bool;
         DBX513_0 : Bool;   // 1;LEV2;HSK13-DPL.CNG.CHECK2-Recoverable error;TK;W0;N;O;M
         DBX513_1 : Bool;   // 1;LEV2;HSK13-DPL.CNG.CHECK2-Error;TK;W0;N;O;M
         DBX513_2 : Bool;   // 1;LEV2;HSK13-DPL.CNG.CHECK2-Time out error;TK;W0;N;O;M
         DBX513_3 : Bool;   // 1;LEV2;HSK13-DPL.CNG.CHECK2-Configuration error;TK;W0;N;O;M
         DBX513_4 : Bool;   // 1;LEV2;HSK13-DPL.CNG.CHECK2-Lock;TK;W0;N;O;M
         DBX513_5 : Bool;
         DBX513_6 : Bool;
         DBX513_7 : Bool;
         DBX514_0 : Bool;   // 1;LEV2;HSK14-DPL.CNG.CHECK3-Recoverable error;TK;W0;N;O;M
         DBX514_1 : Bool;   // 1;LEV2;HSK14-DPL.CNG.CHECK3-Error;TK;W0;N;O;M
         DBX514_2 : Bool;   // 1;LEV2;HSK14-DPL.CNG.CHECK3-Time out error;TK;W0;N;O;M
         DBX514_3 : Bool;   // 1;LEV2;HSK14-DPL.CNG.CHECK3-Configuration error;TK;W0;N;O;M
         DBX514_4 : Bool;   // 1;LEV2;HSK14-DPL.CNG.CHECK3-Lock;TK;W0;N;O;M
         DBX514_5 : Bool;
         DBX514_6 : Bool;
         DBX514_7 : Bool;
         DBX515_0 : Bool;   // 1;LEV2;HSK15-DPL.CNG.CHECK4-Recoverable error;TK;W0;N;O;M
         DBX515_1 : Bool;   // 1;LEV2;HSK15-DPL.CNG.CHECK4-Error;TK;W0;N;O;M
         DBX515_2 : Bool;   // 1;LEV2;HSK15-DPL.CNG.CHECK4-Time out error;TK;W0;N;O;M
         DBX515_3 : Bool;   // 1;LEV2;HSK15-DPL.CNG.CHECK4-Configuration error;TK;W0;N;O;M
         DBX515_4 : Bool;   // 1;LEV2;HSK15-DPL.CNG.CHECK4-Lock;TK;W0;N;O;M
         DBX515_5 : Bool;
         DBX515_6 : Bool;
         DBX515_7 : Bool;
         DBX516_0 : Bool;   // 1;LEV2;HSK16-DPL.CNG.SHFT-Recoverable error;TK;W0;N;O;M
         DBX516_1 : Bool;   // 1;LEV2;HSK16-DPL.CNG.SHFT-Error;TK;W0;N;O;M
         DBX516_2 : Bool;   // 1;LEV2;HSK16-DPL.CNG.SHFT-Time out error;TK;W0;N;O;M
         DBX516_3 : Bool;   // 1;LEV2;HSK16-DPL.CNG.SHFT-Configuration error;TK;W0;N;O;M
         DBX516_4 : Bool;   // 1;LEV2;HSK16-DPL.CNG.SHFT-Lock;TK;W0;N;O;M
         DBX516_5 : Bool;
         DBX516_6 : Bool;
         DBX516_7 : Bool;
         DBX517_0 : Bool;   // 1;LEV2;HSK17-DPL.WAX.BEGIN-Recoverable error;TK;W0;N;O;M
         DBX517_1 : Bool;   // 1;LEV2;HSK17-DPL.WAX.BEGIN-Error;TK;W0;N;O;M
         DBX517_2 : Bool;   // 1;LEV2;HSK17-DPL.WAX.BEGIN-Time out error;TK;W0;N;O;M
         DBX517_3 : Bool;   // 1;LEV2;HSK17-DPL.WAX.BEGIN-Configuration error;TK;W0;N;O;M
         DBX517_4 : Bool;   // 1;LEV2;HSK17-DPL.WAX.BEGIN-Lock;TK;W0;N;O;M
         DBX517_5 : Bool;
         DBX517_6 : Bool;
         DBX517_7 : Bool;
         DBX518_0 : Bool;   // 1;LEV2;HSK18-DPL.WAX.END-Recoverable error;TK;W0;N;O;M
         DBX518_1 : Bool;   // 1;LEV2;HSK18-DPL.WAX.END-Error;TK;W0;N;O;M
         DBX518_2 : Bool;   // 1;LEV2;HSK18-DPL.WAX.END-Time out error;TK;W0;N;O;M
         DBX518_3 : Bool;   // 1;LEV2;HSK18-DPL.WAX.END-Configuration error;TK;W0;N;O;M
         DBX518_4 : Bool;   // 1;LEV2;HSK18-DPL.WAX.END-Lock;TK;W0;N;O;M
         DBX518_5 : Bool;
         DBX518_6 : Bool;
         DBX518_7 : Bool;
         DBX519_0 : Bool;   // 1;LEV2;HSK19-DPL.DMY.LOAD.COAT-Recoverable error;TK;W0;N;O;M
         DBX519_1 : Bool;   // 1;LEV2;HSK19-DPL.DMY.LOAD.COAT-Error;TK;W0;N;O;M
         DBX519_2 : Bool;   // 1;LEV2;HSK19-DPL.DMY.LOAD.COAT-Time out error;TK;W0;N;O;M
         DBX519_3 : Bool;   // 1;LEV2;HSK19-DPL.DMY.LOAD.COAT-Configuration error;TK;W0;N;O;M
         DBX519_4 : Bool;   // 1;LEV2;HSK19-DPL.DMY.LOAD.COAT-Lock;TK;W0;N;O;M
         DBX519_5 : Bool;
         DBX519_6 : Bool;
         DBX519_7 : Bool;
         DBX520_0 : Bool;   // 1;LEV2;HSK20-DPL.DMY.VDI.COAT-Recoverable error;TK;W0;N;O;M
         DBX520_1 : Bool;   // 1;LEV2;HSK20-DPL.DMY.VDI.COAT-Error;TK;W0;N;O;M
         DBX520_2 : Bool;   // 1;LEV2;HSK20-DPL.DMY.VDI.COAT-Time out error;TK;W0;N;O;M
         DBX520_3 : Bool;   // 1;LEV2;HSK20-DPL.DMY.VDI.COAT-Configuration error;TK;W0;N;O;M
         DBX520_4 : Bool;   // 1;LEV2;HSK20-DPL.DMY.VDI.COAT-Lock;TK;W0;N;O;M
         DBX520_5 : Bool;
         DBX520_6 : Bool;
         DBX520_7 : Bool;
         DBX521_0 : Bool;   // 1;LEV2;HSK21-DPL.DMY.COUNT.COAT-Recoverable error;TK;W0;N;O;M
         DBX521_1 : Bool;   // 1;LEV2;HSK21-DPL.DMY.COUNT.COAT-Error;TK;W0;N;O;M
         DBX521_2 : Bool;   // 1;LEV2;HSK21-DPL.DMY.COUNT.COAT-Time out error;TK;W0;N;O;M
         DBX521_3 : Bool;   // 1;LEV2;HSK21-DPL.DMY.COUNT.COAT-Configuration error;TK;W0;N;O;M
         DBX521_4 : Bool;   // 1;LEV2;HSK21-DPL.DMY.COUNT.COAT-Lock;TK;W0;N;O;M
         DBX521_5 : Bool;
         DBX521_6 : Bool;
         DBX521_7 : Bool;
         DBX522_0 : Bool;   // 1;LEV2;HSK22-DPL.R2.OPER-Recoverable error;TK;W0;N;O;M
         DBX522_1 : Bool;   // 1;LEV2;HSK22-DPL.R2.OPER-Error;TK;W0;N;O;M
         DBX522_2 : Bool;   // 1;LEV2;HSK22-DPL.R2.OPER-Time out error;TK;W0;N;O;M
         DBX522_3 : Bool;   // 1;LEV2;HSK22-DPL.R2.OPER-Configuration error;TK;W0;N;O;M
         DBX522_4 : Bool;   // 1;LEV2;HSK22-DPL.R2.OPER-Lock;TK;W0;N;O;M
         DBX522_5 : Bool;
         DBX522_6 : Bool;
         DBX522_7 : Bool;
         DBX523_0 : Bool;   // 1;LEV2;HSK23-DPL.R1.OPER-Recoverable error;TK;W0;N;O;M
         DBX523_1 : Bool;   // 1;LEV2;HSK23-DPL.R1.OPER-Error;TK;W0;N;O;M
         DBX523_2 : Bool;   // 1;LEV2;HSK23-DPL.R1.OPER-Time out error;TK;W0;N;O;M
         DBX523_3 : Bool;   // 1;LEV2;HSK23-DPL.R1.OPER-Configuration error;TK;W0;N;O;M
         DBX523_4 : Bool;   // 1;LEV2;HSK23-DPL.R1.OPER-Lock;TK;W0;N;O;M
         DBX523_5 : Bool;
         DBX523_6 : Bool;
         DBX523_7 : Bool;
         DBX524_0 : Bool;   // 1;LEV2;HSK24-DPL.EXIT.COUNT-Recoverable error;TK;W0;N;O;M
         DBX524_1 : Bool;   // 1;LEV2;HSK24-DPL.EXIT.COUNT-Error;TK;W0;N;O;M
         DBX524_2 : Bool;   // 1;LEV2;HSK24-DPL.EXIT.COUNT-Time out error;TK;W0;N;O;M
         DBX524_3 : Bool;   // 1;LEV2;HSK24-DPL.EXIT.COUNT-Configuration error;TK;W0;N;O;M
         DBX524_4 : Bool;   // 1;LEV2;HSK24-DPL.EXIT.COUNT-Lock;TK;W0;N;O;M
         DBX524_5 : Bool;
         DBX524_6 : Bool;
         DBX524_7 : Bool;
         DBX525_0 : Bool;   // 1;LEV2;HSK25-DPL.INSP.LOAD-Recoverable error;TK;W0;N;O;M
         DBX525_1 : Bool;   // 1;LEV2;HSK25-DPL.INSP.LOAD-Error;TK;W0;N;O;M
         DBX525_2 : Bool;   // 1;LEV2;HSK25-DPL.INSP.LOAD-Time out error;TK;W0;N;O;M
         DBX525_3 : Bool;   // 1;LEV2;HSK25-DPL.INSP.LOAD-Configuration error;TK;W0;N;O;M
         DBX525_4 : Bool;   // 1;LEV2;HSK25-DPL.INSP.LOAD-Lock;TK;W0;N;O;M
         DBX525_5 : Bool;
         DBX525_6 : Bool;
         DBX525_7 : Bool;
         DBX526_0 : Bool;   // 1;LEV2;HSK26-DPL.INSP.VDI-Recoverable error;TK;W0;N;O;M
         DBX526_1 : Bool;   // 1;LEV2;HSK26-DPL.INSP.VDI-Error;TK;W0;N;O;M
         DBX526_2 : Bool;   // 1;LEV2;HSK26-DPL.INSP.VDI-Time out error;TK;W0;N;O;M
         DBX526_3 : Bool;   // 1;LEV2;HSK26-DPL.INSP.VDI-Configuration error;TK;W0;N;O;M
         DBX526_4 : Bool;   // 1;LEV2;HSK26-DPL.INSP.VDI-Lock;TK;W0;N;O;M
         DBX526_5 : Bool;
         DBX526_6 : Bool;
         DBX526_7 : Bool;
